C03582=1013.763,-65.159,-112.589,-25.183,25.961,-41.211
C03583=1013.760,-65.399,-112.570,-25.198,26.028,-41.179
C03584=1013.758,-65.638,-112.552,-25.214,26.096,-41.145
C03585=1013.756,-65.879,-112.533,-25.229,26.164,-41.112
C03586=1013.753,-66.119,-112.513,-25.244,26.231,-41.080
C03587=1013.750,-66.358,-112.495,-25.260,26.301,-41.045
C03588=1013.748,-66.599,-112.475,-25.275,26.369,-41.012
C03589=1013.746,-66.839,-112.456,-25.291,26.439,-40.980
C03590=1013.743,-67.080,-112.437,-25.307,26.508,-40.945
C03591=1013.740,-67.320,-112.417,-25.322,26.578,-40.911
C03592=1013.738,-67.561,-112.398,-25.338,26.649,-40.878
C03593=1013.735,-67.801,-112.379,-25.354,26.720,-40.844
C03594=1013.733,-68.042,-112.360,-25.369,26.790,-40.811
C03595=1013.730,-68.283,-112.341,-25.385,26.862,-40.776
C03596=1013.728,-68.523,-112.322,-25.401,26.933,-40.743
C03597=1013.725,-68.763,-112.303,-25.417,27.006,-40.709
C03598=1013.723,-69.004,-112.283,-25.433,27.078,-40.674
C03599=1013.720,-69.245,-112.264,-25.448,27.151,-40.640
C03600=1013.716,-69.587,-112.236,-25.471,27.255,-40.591
C03601=1013.712,-69.967,-112.206,-25.496,27.371,-40.536
C03602=1013.709,-70.208,-112.187,-25.512,27.446,-40.501
C03603=1013.707,-70.448,-112.167,-25.528,27.520,-40.467
C03604=1013.704,-70.689,-112.149,-25.544,27.595,-40.432
C03605=1013.702,-70.929,-112.130,-25.560,27.669,-40.398
C03606=1013.699,-71.170,-112.111,-25.576,27.746,-40.362
C03607=1013.696,-71.411,-112.091,-25.592,27.821,-40.328
C03608=1013.694,-71.652,-112.072,-25.608,27.897,-40.293
C03609=1013.691,-71.892,-112.053,-25.625,27.974,-40.258
C03610=1013.688,-72.132,-112.034,-25.641,28.052,-40.222
C03611=1013.686,-72.374,-112.014,-25.657,28.128,-40.186
C03612=1013.683,-72.613,-111.996,-25.673,28.205,-40.152
C03613=1013.680,-72.853,-111.976,-25.689,28.283,-40.116
C03614=1013.677,-73.094,-111.957,-25.706,28.362,-40.080
C03615=1013.675,-73.334,-111.938,-25.722,28.440,-40.044
C03616=1013.672,-73.575,-111.919,-25.738,28.519,-40.009
C03617=1013.669,-73.815,-111.900,-25.754,28.598,-39.974
C03618=1013.666,-74.054,-111.881,-25.771,28.678,-39.938
C03619=1013.663,-74.295,-111.861,-25.787,28.757,-39.902
C03620=1013.661,-74.534,-111.842,-25.803,28.838,-39.866
C03621=1013.657,-74.775,-111.823,-25.820,28.919,-39.830
C03622=1013.656,-75.014,-111.804,-25.836,28.999,-39.795
C03623=1013.652,-75.255,-111.784,-25.852,29.081,-39.759
C03624=1013.650,-75.494,-111.765,-25.869,29.162,-39.722
C03625=1013.647,-75.735,-111.746,-25.885,29.244,-39.685
C03626=1013.644,-75.974,-111.727,-25.901,29.326,-39.650
C03627=1013.640,-76.214,-111.708,-25.918,29.409,-39.614
C03628=1013.638,-76.454,-111.690,-25.934,29.492,-39.577
C03629=1013.635,-76.693,-111.670,-25.951,29.575,-39.542
C03630=1013.632,-76.932,-111.651,-25.967,29.659,-39.504
C03631=1013.630,-77.172,-111.632,-25.983,29.742,-39.468
C03632=1013.627,-77.411,-111.612,-26.000,29.827,-39.432
C03633=1013.623,-77.650,-111.594,-26.016,29.911,-39.395
C03634=1013.620,-77.889,-111.574,-26.033,29.996,-39.358
C03635=1013.618,-78.129,-111.556,-26.049,30.081,-39.322
C03636=1013.614,-78.367,-111.536,-26.066,30.167,-39.286
C03637=1013.611,-78.606,-111.517,-26.082,30.252,-39.249
C03638=1013.608,-78.844,-111.498,-26.099,30.339,-39.212
C03639=1013.605,-79.083,-111.479,-26.115,30.425,-39.176
C03640=1013.602,-79.321,-111.460,-26.132,30.511,-39.139
C03641=1013.599,-79.559,-111.441,-26.148,30.598,-39.102
C03642=1013.597,-79.798,-111.422,-26.165,30.686,-39.066
C03643=1013.594,-80.036,-111.403,-26.181,30.772,-39.029
C03644=1013.591,-80.274,-111.384,-26.197,30.861,-38.991
C03645=1013.587,-80.511,-111.365,-26.214,30.949,-38.955
C03646=1013.585,-80.748,-111.346,-26.230,31.038,-38.918
C03647=1013.582,-80.985,-111.327,-26.247,31.125,-38.881
C03648=1013.578,-81.220,-111.308,-26.263,31.215,-38.844
C03649=1013.576,-81.457,-111.289,-26.279,31.303,-38.808
C03650=1013.573,-81.694,-111.270,-26.296,31.393,-38.772
C03651=1013.570,-81.930,-111.251,-26.312,31.483,-38.734
C03652=1013.567,-82.168,-111.233,-26.329,31.573,-38.698
C03653=1013.564,-82.405,-111.213,-26.345,31.664,-38.660
C03654=1013.560,-82.642,-111.195,-26.361,31.755,-38.624
C03655=1013.558,-82.878,-111.176,-26.378,31.846,-38.587
C03656=1013.554,-83.113,-111.157,-26.394,31.937,-38.549
C03657=1013.552,-83.350,-111.138,-26.411,32.029,-38.513
C03658=1013.548,-83.586,-111.119,-26.427,32.121,-38.476
C03659=1013.545,-83.821,-111.101,-26.443,32.213,-38.439
C03660=1013.542,-84.054,-111.082,-26.460,32.304,-38.402
C03661=1013.539,-84.286,-111.063,-26.476,32.396,-38.366
C03662=1013.536,-84.519,-111.044,-26.492,32.488,-38.329
C03663=1013.533,-84.759,-111.025,-26.509,32.584,-38.291
C03664=1013.529,-85.016,-111.004,-26.526,32.686,-38.252
C03665=1013.526,-85.291,-110.983,-26.545,32.796,-38.208
C03666=1013.523,-85.531,-110.963,-26.562,32.893,-38.169
C03667=1013.518,-85.858,-110.937,-26.585,33.025,-38.119
C03668=1013.514,-86.127,-110.915,-26.603,33.135,-38.077
C03669=1013.510,-86.378,-110.895,-26.621,33.237,-38.038
C03670=1013.508,-86.612,-110.877,-26.637,33.332,-38.000
C03671=1013.505,-86.843,-110.858,-26.653,33.428,-37.963
C03672=1013.502,-87.073,-110.840,-26.669,33.523,-37.927
C03673=1013.499,-87.296,-110.822,-26.685,33.614,-37.892
C03674=1013.495,-87.515,-110.804,-26.700,33.705,-37.858
C03675=1013.493,-87.735,-110.787,-26.715,33.797,-37.822
C03676=1013.489,-87.950,-110.769,-26.730,33.886,-37.788
C03677=1013.486,-88.167,-110.753,-26.745,33.978,-37.754
C03678=1013.484,-88.393,-110.735,-26.761,34.073,-37.719
C03679=1013.480,-88.619,-110.716,-26.776,34.168,-37.683
C03680=1013.477,-88.853,-110.697,-26.792,34.267,-37.646
C03681=1013.474,-89.120,-110.676,-26.811,34.380,-37.604
C03682=1013.470,-89.416,-110.652,-26.831,34.506,-37.557
C03683=1013.466,-89.724,-110.627,-26.853,34.638,-37.507
C03684=1013.461,-90.025,-110.603,-26.873,34.768,-37.461
C03685=1013.455,-90.431,-110.571,-26.901,34.943,-37.396
C03686=1013.451,-90.700,-110.549,-26.920,35.060,-37.354
C03687=1013.447,-90.997,-110.525,-26.940,35.190,-37.306
C03688=1013.443,-91.247,-110.505,-26.957,35.298,-37.269
C03689=1013.440,-91.478,-110.486,-26.973,35.401,-37.231
C03690=1013.437,-91.710,-110.467,-26.989,35.502,-37.195
C03691=1013.434,-91.941,-110.449,-27.005,35.604,-37.159
C03692=1013.431,-92.172,-110.430,-27.021,35.707,-37.122
C03693=1013.428,-92.403,-110.412,-27.036,35.809,-37.086
C03694=1013.424,-92.633,-110.393,-27.052,35.911,-37.049
C03695=1013.421,-92.864,-110.375,-27.068,36.014,-37.014
C03696=1013.418,-93.095,-110.356,-27.084,36.118,-36.978
C03697=1013.414,-93.324,-110.338,-27.099,36.220,-36.941
C03698=1013.411,-93.553,-110.319,-27.115,36.324,-36.905
C03699=1013.408,-93.783,-110.300,-27.130,36.427,-36.870
C03700=1013.405,-94.011,-110.282,-27.146,36.531,-36.835
C03701=1013.401,-94.240,-110.263,-27.161,36.635,-36.799
C03702=1013.398,-94.468,-110.245,-27.177,36.738,-36.763
C03703=1013.395,-94.695,-110.227,-27.192,36.843,-36.728
C03704=1013.391,-94.922,-110.208,-27.208,36.947,-36.692
C03705=1013.387,-95.149,-110.190,-27.223,37.051,-36.657
C03706=1013.385,-95.375,-110.172,-27.238,37.156,-36.622
C03707=1013.381,-95.601,-110.153,-27.253,37.259,-36.587
C03708=1013.378,-95.826,-110.135,-27.269,37.365,-36.551
C03709=1013.375,-96.052,-110.117,-27.284,37.469,-36.516
C03710=1013.372,-96.276,-110.100,-27.299,37.574,-36.481
C03711=1013.368,-96.501,-110.081,-27.314,37.678,-36.447
C03712=1013.365,-96.725,-110.062,-27.329,37.784,-36.413
C03713=1013.362,-96.949,-110.045,-27.344,37.888,-36.379
C03714=1013.358,-97.173,-110.026,-27.359,37.995,-36.344
C03715=1013.355,-97.397,-110.008,-27.374,38.100,-36.310
C03716=1013.352,-97.620,-109.990,-27.389,38.207,-36.275
C03717=1013.349,-97.844,-109.973,-27.403,38.312,-36.242
C03718=1013.345,-98.067,-109.955,-27.418,38.419,-36.207
C03719=1013.340,-98.468,-109.922,-27.445,38.610,-36.146
C03720=1013.335,-98.738,-109.900,-27.463,38.739,-36.104
C03721=1013.332,-98.962,-109.882,-27.478,38.848,-36.070
C03722=1013.329,-99.186,-109.864,-27.492,38.955,-36.036
C03723=1013.326,-99.410,-109.846,-27.507,39.064,-36.001
C03724=1013.322,-99.635,-109.827,-27.522,39.173,-35.967
C03725=1013.319,-99.859,-109.809,-27.537,39.283,-35.933
C03726=1013.316,-100.085,-109.791,-27.552,39.393,-35.900
C03727=1013.312,-100.310,-109.773,-27.567,39.504,-35.865
C03728=1013.309,-100.536,-109.754,-27.581,39.613,-35.831
C03729=1013.305,-100.762,-109.736,-27.596,39.725,-35.797
C03730=1013.302,-100.989,-109.717,-27.611,39.836,-35.763
C03731=1013.299,-101.216,-109.700,-27.626,39.949,-35.728
C03732=1013.295,-101.443,-109.681,-27.641,40.061,-35.695
C03733=1013.292,-101.671,-109.662,-27.656,40.174,-35.660
C03734=1013.288,-101.899,-109.643,-27.670,40.288,-35.627
C03735=1013.285,-102.128,-109.624,-27.685,40.402,-35.592
C03736=1013.282,-102.356,-109.607,-27.700,40.517,-35.557
C03737=1013.278,-102.585,-109.588,-27.715,40.632,-35.524
C03738=1013.275,-102.814,-109.569,-27.730,40.746,-35.490
C03739=1013.271,-103.044,-109.551,-27.745,40.862,-35.456
C03740=1013.268,-103.274,-109.532,-27.760,40.979,-35.422
C03741=1013.265,-103.503,-109.513,-27.774,41.095,-35.388
C03742=1013.261,-103.733,-109.494,-27.789,41.212,-35.354
C03743=1013.257,-103.964,-109.475,-27.804,41.329,-35.321
C03744=1013.253,-104.194,-109.457,-27.819,41.447,-35.287
C03745=1013.251,-104.425,-109.438,-27.834,41.565,-35.253
C03746=1013.247,-104.655,-109.420,-27.848,41.683,-35.219
C03747=1013.243,-104.887,-109.400,-27.863,41.802,-35.187
C03748=1013.241,-105.118,-109.381,-27.878,41.921,-35.152
C03749=1013.236,-105.349,-109.362,-27.893,42.041,-35.119
C03750=1013.233,-105.580,-109.344,-27.907,42.161,-35.086
C03751=1013.230,-105.812,-109.324,-27.922,42.281,-35.052
C03752=1013.226,-106.043,-109.306,-27.937,42.402,-35.019
C03753=1013.222,-106.275,-109.287,-27.952,42.522,-34.986
C03754=1013.219,-106.510,-109.268,-27.966,42.645,-34.953
C03755=1013.216,-106.752,-109.248,-27.982,42.772,-34.918
C03756=1013.212,-107.005,-109.227,-27.998,42.904,-34.883
C03757=1013.207,-107.267,-109.206,-28.014,43.043,-34.846
C03758=1013.204,-107.537,-109.184,-28.031,43.186,-34.806
C03759=1013.199,-107.812,-109.161,-28.049,43.332,-34.767
C03760=1013.195,-108.089,-109.138,-28.066,43.478,-34.728
C03761=1013.191,-108.362,-109.117,-28.083,43.625,-34.690
C03762=1013.187,-108.631,-109.095,-28.100,43.769,-34.652
C03763=1013.183,-108.891,-109.074,-28.116,43.908,-34.616
C03764=1013.180,-109.142,-109.053,-28.132,44.042,-34.581
C03765=1013.176,-109.383,-109.033,-28.147,44.172,-34.548
C03766=1013.170,-109.734,-109.003,-28.169,44.360,-34.500
C03767=1013.165,-110.079,-108.975,-28.190,44.548,-34.453
C03768=1013.162,-110.311,-108.957,-28.205,44.674,-34.422
C03769=1013.158,-110.542,-108.938,-28.219,44.800,-34.391
C03770=1013.155,-110.773,-108.919,-28.233,44.927,-34.359
C03771=1013.151,-111.005,-108.900,-28.248,45.053,-34.328
C03772=1013.148,-111.236,-108.881,-28.262,45.180,-34.296
C03773=1013.144,-111.468,-108.862,-28.276,45.307,-34.265
C03774=1013.140,-111.698,-108.843,-28.290,45.433,-34.235
C03775=1013.137,-111.930,-108.823,-28.305,45.561,-34.204
C03776=1013.134,-112.162,-108.805,-28.319,45.690,-34.174
C03777=1013.129,-112.393,-108.786,-28.333,45.818,-34.142
C03778=1013.126,-112.624,-108.767,-28.347,45.947,-34.112
C03779=1013.123,-112.855,-108.747,-28.362,46.074,-34.082
C03780=1013.119,-113.087,-108.729,-28.376,46.205,-34.052
C03781=1013.116,-113.318,-108.709,-28.390,46.334,-34.021
C03782=1013.112,-113.549,-108.691,-28.404,46.462,-33.992
C03783=1013.109,-113.781,-108.671,-28.418,46.593,-33.962
C03784=1013.106,-114.011,-108.652,-28.433,46.723,-33.932
C03785=1013.102,-114.243,-108.633,-28.447,46.853,-33.903
C03786=1013.098,-114.474,-108.614,-28.461,46.984,-33.872
C03787=1013.095,-114.705,-108.595,-28.475,47.115,-33.843
C03788=1013.092,-114.937,-108.576,-28.489,47.247,-33.814
C03789=1013.088,-115.168,-108.557,-28.503,47.378,-33.785
C03790=1013.085,-115.399,-108.538,-28.517,47.510,-33.756
C03791=1013.081,-115.630,-108.519,-28.531,47.641,-33.728
C03792=1013.077,-115.861,-108.499,-28.545,47.773,-33.699
C03793=1013.074,-116.093,-108.481,-28.559,47.905,-33.670
C03794=1013.071,-116.324,-108.461,-28.573,48.038,-33.642
C03795=1013.066,-116.555,-108.442,-28.587,48.171,-33.614
C03796=1013.064,-116.786,-108.424,-28.601,48.304,-33.584
C03797=1013.060,-117.017,-108.404,-28.615,48.437,-33.557
C03798=1013.057,-117.248,-108.385,-28.629,48.570,-33.530
C03799=1013.053,-117.479,-108.365,-28.643,48.704,-33.501
C03800=1013.050,-117.711,-108.346,-28.657,48.837,-33.474
C03801=1013.046,-117.942,-108.328,-28.671,48.972,-33.446
C03802=1013.043,-118.173,-108.308,-28.685,49.107,-33.419
C03803=1013.040,-118.404,-108.290,-28.699,49.240,-33.393
C03804=1013.036,-118.635,-108.270,-28.713,49.376,-33.366
C03805=1013.033,-118.867,-108.251,-28.727,49.510,-33.339
C03806=1013.029,-119.097,-108.232,-28.741,49.646,-33.311
C03807=1013.023,-119.517,-108.197,-28.767,49.892,-33.263
C03808=1013.019,-119.791,-108.174,-28.783,50.052,-33.234
C03809=1013.016,-120.021,-108.155,-28.797,50.188,-33.207
C03810=1013.012,-120.253,-108.135,-28.811,50.324,-33.182
C03811=1013.009,-120.484,-108.117,-28.825,50.460,-33.156
C03812=1013.005,-120.715,-108.098,-28.839,50.597,-33.130
C03813=1013.001,-120.946,-108.078,-28.853,50.734,-33.104
C03814=1012.998,-121.177,-108.059,-28.867,50.871,-33.080
C03815=1012.995,-121.408,-108.039,-28.881,51.009,-33.055
C03816=1012.992,-121.639,-108.021,-28.895,51.146,-33.030
C03817=1012.988,-121.871,-108.001,-28.909,51.283,-33.005
C03818=1012.985,-122.101,-107.982,-28.923,51.421,-32.981
C03819=1012.982,-122.333,-107.962,-28.937,51.560,-32.957
C03820=1012.978,-122.563,-107.944,-28.951,51.697,-32.933
C03821=1012.974,-122.794,-107.924,-28.965,51.836,-32.909
C03822=1012.971,-123.025,-107.906,-28.979,51.974,-32.885
C03823=1012.968,-123.257,-107.886,-28.993,52.113,-32.862
C03824=1012.965,-123.487,-107.867,-29.007,52.253,-32.839
C03825=1012.962,-123.718,-107.848,-29.021,52.392,-32.815
C03826=1012.958,-123.949,-107.828,-29.035,52.531,-32.792
C03827=1012.955,-124.180,-107.809,-29.050,52.671,-32.770
C03828=1012.951,-124.411,-107.789,-29.064,52.811,-32.747
C03829=1012.949,-124.642,-107.771,-29.078,52.950,-32.725
C03830=1012.945,-124.874,-107.751,-29.092,53.091,-32.702
C03831=1012.942,-125.104,-107.732,-29.107,53.231,-32.681
C03832=1012.938,-125.336,-107.712,-29.121,53.372,-32.658
C03833=1012.935,-125.566,-107.693,-29.135,53.512,-32.638
C03834=1012.932,-125.797,-107.674,-29.149,53.654,-32.616
C03835=1012.929,-126.028,-107.654,-29.164,53.795,-32.595
C03836=1012.926,-126.259,-107.635,-29.178,53.936,-32.573
C03837=1012.922,-126.490,-107.615,-29.193,54.078,-32.552
C03838=1012.919,-126.721,-107.596,-29.207,54.219,-32.532
C03839=1012.916,-126.952,-107.578,-29.221,54.362,-32.511
C03840=1012.913,-127.183,-107.558,-29.236,54.504,-32.491
C03841=1012.910,-127.414,-107.539,-29.251,54.646,-32.472
C03842=1012.906,-127.645,-107.519,-29.265,54.789,-32.451
C03843=1012.903,-127.876,-107.500,-29.280,54.931,-32.432
C03844=1012.900,-128.106,-107.481,-29.294,55.074,-32.412
C03845=1012.896,-128.337,-107.461,-29.309,55.218,-32.393
C03846=1012.890,-128.749,-107.427,-29.336,55.474,-32.360
C03847=1012.886,-129.030,-107.403,-29.354,55.649,-32.337
C03848=1012.883,-129.261,-107.384,-29.369,55.792,-32.319
C03849=1012.880,-129.491,-107.365,-29.384,55.936,-32.301
C03850=1012.877,-129.722,-107.345,-29.399,56.081,-32.283
C03851=1012.874,-129.953,-107.326,-29.414,56.225,-32.266
C03852=1012.871,-130.184,-107.307,-29.429,56.370,-32.248
C03853=1012.867,-130.415,-107.287,-29.444,56.515,-32.230
C03854=1012.865,-130.646,-107.267,-29.460,56.659,-32.215
C03855=1012.862,-130.876,-107.248,-29.475,56.805,-32.198
C03856=1012.858,-131.108,-107.228,-29.490,56.950,-32.182
C03857=1012.855,-131.339,-107.210,-29.506,57.095,-32.165
C03858=1012.852,-131.570,-107.191,-29.521,57.242,-32.148
C03859=1012.849,-131.800,-107.171,-29.537,57.388,-32.133
C03860=1012.846,-132.031,-107.152,-29.553,57.534,-32.118
C03861=1012.843,-132.262,-107.132,-29.568,57.680,-32.102
C03862=1012.840,-132.493,-107.113,-29.585,57.827,-32.089
C03863=1012.837,-132.724,-107.093,-29.600,57.974,-32.073
C03864=1012.834,-132.955,-107.074,-29.616,58.121,-32.059
C03865=1012.830,-133.185,-107.055,-29.633,58.268,-32.045
C03866=1012.828,-133.416,-107.035,-29.649,58.415,-32.031
C03867=1012.825,-133.647,-107.016,-29.665,58.563,-32.017
C03868=1012.821,-133.878,-106.996,-29.682,58.710,-32.004
C03869=1012.818,-134.109,-106.977,-29.698,58.858,-31.992
C03870=1013.073,-134.133,-107.391,-28.594,48.007,-33.824
C03871=1013.076,-133.902,-107.411,-28.577,47.850,-33.859
C03872=1013.080,-133.672,-107.430,-28.560,47.694,-33.892
C03873=1013.084,-133.441,-107.449,-28.544,47.538,-33.928
C03874=1013.089,-133.210,-107.468,-28.527,47.382,-33.964
C03875=1013.093,-132.979,-107.487,-28.510,47.227,-33.999
C03876=1013.096,-132.748,-107.506,-28.493,47.070,-34.035
C03877=1013.101,-132.517,-107.525,-28.476,46.914,-34.071
C03878=1013.105,-132.286,-107.544,-28.458,46.759,-34.107
C03879=1013.109,-132.055,-107.563,-28.441,46.604,-34.143
C03880=1013.114,-131.824,-107.582,-28.424,46.448,-34.181
C03881=1013.118,-131.594,-107.600,-28.407,46.294,-34.218
C03882=1013.121,-131.363,-107.620,-28.390,46.139,-34.254
C03883=1013.126,-131.132,-107.639,-28.373,45.985,-34.291
C03884=1013.130,-130.901,-107.658,-28.355,45.831,-34.329
C03885=1013.134,-130.670,-107.677,-28.338,45.677,-34.367
C03886=1013.138,-130.439,-107.696,-28.321,45.524,-34.405
C03887=1013.143,-130.208,-107.715,-28.303,45.371,-34.442
C03888=1013.147,-129.977,-107.734,-28.286,45.217,-34.481
C03889=1013.151,-129.746,-107.753,-28.268,45.064,-34.520
C03890=1013.155,-129.516,-107.771,-28.251,44.911,-34.558
C03891=1013.159,-129.285,-107.791,-28.233,44.759,-34.598
C03892=1013.163,-129.054,-107.810,-28.215,44.606,-34.636
C03893=1013.171,-128.685,-107.841,-28.187,44.364,-34.699
C03894=1013.176,-128.361,-107.867,-28.162,44.152,-34.754
C03895=1013.180,-128.130,-107.886,-28.144,43.999,-34.795
C03896=1013.184,-127.899,-107.905,-28.127,43.849,-34.834
C03897=1013.189,-127.668,-107.924,-28.109,43.698,-34.875
C03898=1013.193,-127.437,-107.943,-28.091,43.548,-34.916
C03899=1013.198,-127.207,-107.962,-28.073,43.398,-34.957
C03900=1013.202,-126.976,-107.981,-28.055,43.247,-34.998
C03901=1013.206,-126.745,-108.000,-28.037,43.098,-35.039
C03902=1013.210,-126.514,-108.018,-28.018,42.948,-35.081
C03903=1013.214,-126.283,-108.037,-28.000,42.798,-35.122
C03904=1013.219,-126.052,-108.056,-27.982,42.649,-35.163
C03905=1013.223,-125.821,-108.074,-27.964,42.500,-35.206
C03906=1013.227,-125.590,-108.093,-27.945,42.352,-35.248
C03907=1013.232,-125.359,-108.112,-27.927,42.203,-35.289
C03908=1013.236,-125.128,-108.132,-27.908,42.056,-35.332
C03909=1013.240,-124.897,-108.150,-27.890,41.907,-35.375
C03910=1013.244,-124.666,-108.169,-27.871,41.759,-35.417
C03911=1013.249,-124.435,-108.188,-27.852,41.612,-35.461
C03912=1013.253,-124.204,-108.207,-27.833,41.464,-35.504
C03913=1013.258,-123.973,-108.225,-27.815,41.318,-35.547
C03914=1013.262,-123.742,-108.244,-27.796,41.171,-35.591
C03915=1013.267,-123.511,-108.263,-27.777,41.025,-35.634
C03916=1013.271,-123.280,-108.282,-27.758,40.879,-35.679
C03917=1013.275,-123.049,-108.301,-27.739,40.733,-35.722
C03918=1013.279,-122.818,-108.319,-27.720,40.587,-35.766
C03919=1013.283,-122.587,-108.338,-27.701,40.441,-35.812
C03920=1013.288,-122.356,-108.357,-27.681,40.296,-35.856
C03921=1013.292,-122.125,-108.376,-27.662,40.151,-35.900
C03922=1013.296,-121.894,-108.395,-27.643,40.006,-35.946
C03923=1013.300,-121.663,-108.413,-27.623,39.862,-35.991
C03924=1013.305,-121.432,-108.431,-27.604,39.718,-36.037
C03925=1013.310,-121.201,-108.450,-27.584,39.573,-36.082
C03926=1013.314,-120.970,-108.469,-27.565,39.430,-36.127
C03927=1013.318,-120.738,-108.488,-27.545,39.287,-36.173
C03928=1013.323,-120.507,-108.507,-27.525,39.144,-36.219
C03929=1013.327,-120.276,-108.526,-27.505,39.000,-36.265
C03930=1013.331,-120.045,-108.545,-27.486,38.858,-36.311
C03931=1013.335,-119.814,-108.563,-27.466,38.715,-36.359
C03932=1013.340,-119.569,-108.582,-27.444,38.565,-36.407
C03933=1013.344,-119.353,-108.600,-27.425,38.432,-36.452
C03934=1013.348,-119.121,-108.618,-27.405,38.290,-36.498
C03935=1013.353,-118.890,-108.637,-27.385,38.149,-36.546
C03936=1013.357,-118.659,-108.656,-27.365,38.008,-36.593
C03937=1013.361,-118.428,-108.675,-27.344,37.867,-36.641
C03938=1013.366,-118.197,-108.694,-27.324,37.726,-36.689
C03939=1013.371,-117.966,-108.712,-27.304,37.586,-36.736
C03940=1013.375,-117.734,-108.730,-27.283,37.446,-36.784
C03941=1013.379,-117.503,-108.749,-27.262,37.306,-36.833
C03942=1013.384,-117.272,-108.768,-27.242,37.166,-36.881
C03943=1013.388,-117.041,-108.787,-27.221,37.027,-36.930
C03944=1013.392,-116.810,-108.806,-27.200,36.887,-36.978
C03945=1013.396,-116.578,-108.824,-27.179,36.749,-37.026
C03946=1013.401,-116.347,-108.842,-27.158,36.611,-37.075
C03947=1013.406,-116.116,-108.861,-27.137,36.473,-37.124
C03948=1013.410,-115.885,-108.880,-27.116,36.335,-37.173
C03949=1013.414,-115.654,-108.899,-27.095,36.197,-37.223
C03950=1013.418,-115.422,-108.917,-27.073,36.059,-37.272
C03951=1013.423,-115.191,-108.936,-27.052,35.922,-37.322
C03952=1013.427,-114.960,-108.954,-27.031,35.785,-37.372
C03953=1013.432,-114.729,-108.973,-27.009,35.649,-37.422
C03954=1013.436,-114.497,-108.991,-26.988,35.512,-37.472
C03955=1013.440,-114.266,-109.010,-26.966,35.376,-37.523
C03956=1013.444,-114.035,-109.028,-26.944,35.241,-37.573
C03957=1013.449,-113.804,-109.047,-26.923,35.105,-37.623
C03958=1013.453,-113.572,-109.065,-26.901,34.970,-37.674
C03959=1013.458,-113.341,-109.084,-26.879,34.835,-37.726
C03960=1013.462,-113.110,-109.102,-26.857,34.700,-37.777
C03961=1013.466,-112.878,-109.121,-26.835,34.566,-37.828
C03962=1013.470,-112.647,-109.140,-26.813,34.432,-37.879
C03963=1013.474,-112.416,-109.158,-26.791,34.299,-37.930
C03964=1013.480,-112.185,-109.176,-26.768,34.165,-37.981
C03965=1013.484,-111.953,-109.195,-26.746,34.031,-38.034
C03966=1013.488,-111.722,-109.213,-26.723,33.899,-38.085
C03967=1013.492,-111.491,-109.232,-26.701,33.766,-38.138
C03968=1013.496,-111.259,-109.250,-26.678,33.635,-38.189
C03969=1013.501,-111.028,-109.269,-26.656,33.502,-38.241
C03970=1013.505,-110.797,-109.287,-26.633,33.372,-38.293
C03971=1013.509,-110.565,-109.305,-26.611,33.240,-38.346
C03972=1013.513,-110.351,-109.322,-26.589,33.119,-38.395
C03973=1013.517,-110.137,-109.340,-26.568,32.999,-38.443
C03974=1013.522,-109.871,-109.361,-26.542,32.849,-38.503
C03975=1013.526,-109.639,-109.379,-26.519,32.719,-38.556
C03976=1013.531,-109.406,-109.397,-26.496,32.588,-38.610
C03977=1013.535,-109.165,-109.416,-26.472,32.454,-38.664
C03978=1013.540,-108.915,-109.437,-26.447,32.315,-38.720
C03979=1013.545,-108.654,-109.458,-26.421,32.171,-38.781
C03980=1013.550,-108.386,-109.478,-26.394,32.022,-38.843
C03981=1013.555,-108.112,-109.500,-26.366,31.871,-38.907
C03982=1013.560,-107.835,-109.522,-26.338,31.720,-38.971
C03983=1013.565,-107.560,-109.545,-26.310,31.568,-39.036
C03984=1013.570,-107.290,-109.566,-26.282,31.421,-39.099
C03985=1013.575,-107.028,-109.587,-26.256,31.278,-39.161
C03986=1013.580,-106.775,-109.606,-26.230,31.141,-39.219
C03987=1013.584,-106.533,-109.626,-26.205,31.010,-39.275
C03988=1013.588,-106.298,-109.644,-26.181,30.883,-39.330
C03989=1013.593,-106.067,-109.663,-26.157,30.758,-39.385
C03990=1013.597,-105.835,-109.682,-26.133,30.634,-39.438
C03991=1013.601,-105.604,-109.699,-26.109,30.510,-39.493
C03992=1013.605,-105.372,-109.718,-26.085,30.387,-39.547
C03993=1013.610,-105.140,-109.736,-26.061,30.263,-39.602
C03994=1013.614,-104.909,-109.755,-26.036,30.141,-39.657
C03995=1013.618,-104.679,-109.772,-26.012,30.020,-39.711
C03996=1013.623,-104.448,-109.791,-25.988,29.898,-39.766
C03997=1013.626,-104.217,-109.809,-25.964,29.777,-39.821
C03998=1013.630,-103.987,-109.827,-25.940,29.655,-39.875
C03999=1013.634,-103.757,-109.846,-25.915,29.535,-39.930
C04000=1013.639,-103.527,-109.864,-25.891,29.415,-39.985
C04001=1013.643,-103.297,-109.882,-25.867,29.296,-40.040
C04002=1013.647,-103.066,-109.900,-25.842,29.177,-40.095
C04003=1013.651,-102.837,-109.918,-25.817,29.057,-40.150
C04004=1013.656,-102.607,-109.936,-25.793,28.940,-40.205
C04005=1013.660,-102.379,-109.955,-25.769,28.822,-40.260
C04006=1013.664,-102.149,-109.972,-25.744,28.705,-40.315
C04007=1013.667,-101.921,-109.990,-25.719,28.588,-40.370
C04008=1013.672,-101.693,-110.008,-25.695,28.472,-40.424
C04009=1013.676,-101.465,-110.026,-25.670,28.356,-40.480
C04010=1013.681,-101.238,-110.044,-25.646,28.241,-40.535
C04011=1013.684,-101.011,-110.062,-25.621,28.126,-40.590
C04012=1013.688,-100.785,-110.080,-25.596,28.013,-40.644
C04013=1013.692,-100.559,-110.097,-25.572,27.899,-40.700
C04014=1013.696,-100.332,-110.115,-25.547,27.786,-40.754
C04015=1013.700,-100.107,-110.133,-25.523,27.673,-40.809
C04016=1013.704,-99.881,-110.151,-25.498,27.562,-40.863
C04017=1013.708,-99.657,-110.168,-25.473,27.450,-40.918
C04018=1013.713,-99.373,-110.190,-25.442,27.310,-40.986
C04019=1013.720,-98.984,-110.221,-25.399,27.119,-41.081
C04020=1013.724,-98.760,-110.238,-25.375,27.008,-41.136
C04021=1013.728,-98.537,-110.256,-25.350,26.900,-41.190
C04022=1013.731,-98.312,-110.274,-25.325,26.790,-41.245
C04023=1013.735,-98.089,-110.292,-25.300,26.682,-41.299
C04024=1013.739,-97.865,-110.309,-25.276,26.574,-41.354
C04025=1013.744,-97.642,-110.327,-25.251,26.466,-41.408
C04026=1013.747,-97.419,-110.344,-25.226,26.358,-41.463
C04027=1013.751,-97.195,-110.361,-25.201,26.251,-41.518
C04028=1013.754,-96.971,-110.379,-25.176,26.144,-41.574
C04029=1013.759,-96.747,-110.397,-25.151,26.037,-41.627
C04030=1013.763,-96.523,-110.414,-25.125,25.931,-41.683
C04031=1013.767,-96.298,-110.432,-25.100,25.825,-41.738
C04032=1013.770,-96.073,-110.449,-25.075,25.719,-41.793
C04033=1013.774,-95.849,-110.467,-25.050,25.613,-41.848
C04034=1013.778,-95.622,-110.484,-25.024,25.507,-41.904
C04035=1013.782,-95.397,-110.502,-24.999,25.402,-41.959
C04036=1013.786,-95.171,-110.520,-24.973,25.296,-42.016
C04037=1013.790,-94.944,-110.537,-24.947,25.191,-42.071
C04038=1013.793,-94.716,-110.555,-24.921,25.086,-42.128
C04039=1013.797,-94.489,-110.572,-24.896,24.980,-42.183
C04040=1013.801,-94.261,-110.591,-24.870,24.875,-42.241
C04041=1013.805,-94.033,-110.609,-24.844,24.771,-42.296
C04042=1013.809,-93.804,-110.627,-24.818,24.667,-42.352
C04043=1013.813,-93.574,-110.644,-24.791,24.562,-42.410
C04044=1013.817,-93.345,-110.662,-24.765,24.458,-42.466
C04045=1013.820,-93.116,-110.680,-24.739,24.355,-42.523
C04046=1013.824,-92.886,-110.698,-24.713,24.251,-42.579
C04047=1013.828,-92.655,-110.716,-24.686,24.147,-42.636
C04048=1013.832,-92.424,-110.735,-24.659,24.044,-42.695
C04049=1013.836,-92.194,-110.752,-24.633,23.941,-42.752
C04050=1013.839,-91.963,-110.770,-24.607,23.839,-42.808
C04051=1013.843,-91.731,-110.788,-24.580,23.736,-42.865
C04052=1013.847,-91.500,-110.806,-24.553,23.634,-42.923
C04053=1013.851,-91.269,-110.825,-24.526,23.532,-42.981
C04054=1013.855,-91.018,-110.844,-24.498,23.423,-43.041
C04055=1013.859,-90.722,-110.867,-24.463,23.293,-43.117
C04056=1013.864,-90.453,-110.889,-24.432,23.175,-43.183
C04057=1013.870,-90.047,-110.919,-24.385,23.001,-43.283
C04058=1013.876,-89.746,-110.943,-24.350,22.872,-43.358
C04059=1013.880,-89.438,-110.967,-24.314,22.739,-43.434
C04060=1013.885,-89.142,-110.990,-24.279,22.614,-43.508
C04061=1013.889,-88.874,-111.011,-24.248,22.500,-43.574
C04062=1013.893,-88.641,-111.029,-24.221,22.402,-43.632
C04063=1013.897,-88.414,-111.047,-24.194,22.306,-43.688
C04064=1013.900,-88.188,-111.065,-24.168,22.211,-43.744
C04065=1013.904,-87.971,-111.082,-24.142,22.121,-43.798
C04066=1013.921,-86.931,-111.162,-24.009,21.652,-44.080
C04067=1013.925,-86.605,-111.188,-24.010,21.651,-44.075
C04068=1013.931,-86.261,-111.214,-24.011,21.651,-44.069
C04069=1013.934,-86.030,-111.232,-24.011,21.650,-44.065
C04070=1013.938,-85.785,-111.251,-24.012,21.650,-44.062
C04071=1013.941,-85.529,-111.271,-24.012,21.649,-44.060
C04072=1013.945,-85.276,-111.291,-24.012,21.650,-44.056
C04073=1013.949,-85.034,-111.309,-24.013,21.649,-44.053
C04074=1013.952,-84.812,-111.327,-24.013,21.649,-44.049
C04075=1013.958,-84.404,-111.359,-24.014,21.648,-44.043
C04076=1013.964,-84.005,-111.390,-24.015,21.648,-44.036
C04077=1013.970,-83.604,-111.421,-24.016,21.647,-44.031
C04078=1013.977,-83.204,-111.452,-24.016,21.646,-44.025
C04079=1013.982,-82.801,-111.484,-24.017,21.645,-44.019
C04080=1013.988,-82.399,-111.515,-24.018,21.644,-44.014
C04081=1013.993,-81.997,-111.546,-24.019,21.644,-44.007
C04082=1013.999,-81.593,-111.578,-24.020,21.643,-44.001
C04083=1014.004,-81.189,-111.609,-24.020,21.643,-43.995
C04084=1014.010,-80.784,-111.641,-24.021,21.642,-43.990
C04085=1014.015,-80.379,-111.672,-24.022,21.641,-43.984
C04086=1014.021,-79.973,-111.704,-24.023,21.641,-43.977
C04087=1014.026,-79.567,-111.736,-24.023,21.640,-43.972
C04088=1014.032,-79.160,-111.767,-24.024,21.639,-43.966
C04089=1014.038,-78.753,-111.799,-24.025,21.638,-43.960
C04090=1014.043,-78.345,-111.830,-24.026,21.638,-43.953
C04091=1014.048,-77.937,-111.863,-24.027,21.637,-43.948
C04092=1014.053,-77.529,-111.894,-24.027,21.637,-43.942
C04093=1014.059,-77.120,-111.926,-24.028,21.636,-43.936
C04094=1014.063,-76.710,-111.958,-24.029,21.636,-43.929
C04095=1014.069,-76.301,-111.990,-24.030,21.635,-43.924
C04096=1014.074,-75.891,-112.022,-24.031,21.634,-43.918
C04097=1014.079,-75.481,-112.053,-24.031,21.633,-43.912
C04098=1014.085,-75.072,-112.086,-24.032,21.633,-43.905
C04099=1014.089,-74.660,-112.118,-24.033,21.632,-43.900
C04100=1014.094,-74.250,-112.150,-24.034,21.632,-43.894
C04101=1014.099,-73.839,-112.183,-24.034,21.631,-43.888
C04102=1014.104,-73.429,-112.215,-24.035,21.631,-43.881
C04103=1014.109,-73.018,-112.246,-24.036,21.630,-43.876
C04104=1014.114,-72.607,-112.278,-24.037,21.629,-43.870
C04105=1014.118,-72.196,-112.311,-24.038,21.628,-43.865
C04106=1014.123,-71.785,-112.343,-24.039,21.627,-43.857
C04107=1014.128,-71.374,-112.376,-24.039,21.626,-43.851
C04108=1014.132,-70.962,-112.407,-24.040,21.626,-43.846
C04109=1014.137,-70.552,-112.440,-24.041,21.625,-43.839
C04110=1014.141,-70.141,-112.471,-24.042,21.625,-43.833
C04111=1014.146,-69.730,-112.504,-24.042,21.624,-43.827
C04112=1014.150,-69.318,-112.536,-24.043,21.623,-43.822
C04113=1014.155,-68.908,-112.568,-24.044,21.623,-43.815
C04114=1014.159,-68.498,-112.601,-24.045,21.622,-43.809
C04115=1014.163,-68.086,-112.633,-24.046,21.621,-43.804
C04116=1014.167,-67.677,-112.665,-24.046,21.621,-43.798
C04117=1014.171,-67.266,-112.698,-24.047,21.620,-43.791
C04118=1014.176,-66.856,-112.729,-24.048,21.620,-43.785
C04119=1014.180,-66.448,-112.761,-24.049,21.619,-43.780
C04120=1014.184,-66.037,-112.794,-24.049,21.618,-43.774
C04121=1014.188,-65.629,-112.826,-24.050,21.617,-43.768
C04122=1014.192,-65.221,-112.858,-24.051,21.617,-43.761
C04123=1014.196,-64.812,-112.890,-24.052,21.616,-43.756
C04124=1014.200,-64.404,-112.922,-24.053,21.615,-43.750
C04125=1014.204,-63.997,-112.955,-24.053,21.615,-43.744
C04126=1014.207,-63.590,-112.986,-24.054,21.615,-43.737
C04127=1014.212,-63.184,-113.019,-24.055,21.614,-43.732
C04128=1014.215,-62.778,-113.051,-24.056,21.613,-43.726
C04129=1014.219,-62.373,-113.083,-24.057,21.612,-43.720
C04130=1014.222,-61.968,-113.115,-24.057,21.611,-43.715
C04131=1014.226,-61.564,-113.146,-24.058,21.611,-43.708
C04132=1014.229,-61.159,-113.178,-24.059,21.610,-43.702
C04133=1014.233,-60.756,-113.210,-24.060,21.610,-43.697
C04134=1014.237,-60.354,-113.242,-24.061,21.610,-43.691
C04135=1014.240,-59.952,-113.273,-24.061,21.609,-43.686
C04136=1014.244,-59.551,-113.305,-24.062,21.608,-43.680
C04137=1014.247,-59.150,-113.337,-24.063,21.608,-43.673
C04138=1014.250,-58.750,-113.369,-24.064,21.607,-43.667
C04139=1014.254,-58.350,-113.400,-24.064,21.606,-43.662
C04140=1014.257,-57.951,-113.432,-24.065,21.606,-43.656
C04141=1014.260,-57.552,-113.463,-24.066,21.605,-43.651
C04142=1014.264,-57.154,-113.495,-24.067,21.604,-43.645
C04143=1014.267,-56.755,-113.526,-24.067,21.603,-43.639
C04144=1014.270,-56.358,-113.558,-24.068,21.603,-43.632
C04145=1014.273,-55.960,-113.589,-24.069,21.602,-43.627
C04146=1014.276,-55.562,-113.621,-24.070,21.603,-43.621
C04147=1014.279,-55.166,-113.653,-24.071,21.602,-43.616
C04148=1014.282,-54.768,-113.684,-24.071,21.601,-43.610
C04149=1014.285,-54.371,-113.715,-24.072,21.600,-43.604
C04150=1014.288,-53.974,-113.748,-24.073,21.599,-43.599
C04151=1014.290,-53.578,-113.779,-24.073,21.599,-43.593
C04152=1014.293,-53.180,-113.810,-24.074,21.598,-43.588
C04153=1014.296,-52.784,-113.842,-24.075,21.598,-43.581
C04154=1014.299,-52.386,-113.873,-24.076,21.598,-43.575
C04155=1014.302,-51.989,-113.905,-24.077,21.597,-43.570
C04156=1014.305,-51.593,-113.936,-24.077,21.596,-43.564
C04157=1014.307,-51.196,-113.968,-24.078,21.595,-43.558
C04158=1014.310,-50.799,-114.000,-24.079,21.595,-43.553
C04159=1014.313,-50.402,-114.032,-24.080,21.594,-43.547
C04160=1014.315,-50.004,-114.063,-24.080,21.593,-43.542
C04161=1014.317,-49.607,-114.095,-24.081,21.592,-43.536
C04162=1014.320,-49.211,-114.127,-24.082,21.592,-43.531
C04163=1014.323,-48.813,-114.158,-24.083,21.592,-43.525
C04164=1014.325,-48.416,-114.190,-24.084,21.592,-43.518
C04165=1014.328,-48.018,-114.221,-24.084,21.591,-43.512
C04166=1014.330,-47.622,-114.254,-24.085,21.590,-43.507
C04167=1014.333,-47.225,-114.285,-24.086,21.589,-43.501
C04168=1014.335,-46.827,-114.317,-24.086,21.588,-43.496
C04169=1014.338,-46.430,-114.348,-24.087,21.589,-43.490
C04170=1014.340,-46.033,-114.381,-24.088,21.588,-43.485
C04171=1014.341,-45.636,-114.413,-24.089,21.587,-43.479
C04172=1014.344,-45.238,-114.444,-24.089,21.586,-43.473
C04173=1014.346,-44.841,-114.476,-24.090,21.585,-43.468
C04174=1014.349,-44.443,-114.508,-24.091,21.585,-43.462
C04175=1014.350,-44.047,-114.540,-24.092,21.585,-43.457
C04176=1014.352,-43.649,-114.572,-24.092,21.584,-43.451
C04177=1014.355,-43.252,-114.604,-24.093,21.584,-43.444
C04178=1014.357,-42.854,-114.636,-24.094,21.583,-43.439
C04179=1014.359,-42.457,-114.667,-24.095,21.582,-43.433
C04180=1014.361,-42.060,-114.700,-24.096,21.582,-43.427
C04181=1014.363,-41.663,-114.732,-24.096,21.582,-43.422
C04182=1014.365,-41.266,-114.763,-24.097,21.581,-43.417
C04183=1014.367,-40.868,-114.795,-24.098,21.580,-43.411
C04184=1014.368,-40.470,-114.828,-24.099,21.579,-43.405
C04185=1014.370,-40.073,-114.859,-24.099,21.579,-43.400
C04186=1014.372,-39.676,-114.892,-24.100,21.578,-43.394
C04187=1014.375,-39.279,-114.924,-24.101,21.578,-43.389
C04188=1014.376,-38.882,-114.956,-24.102,21.577,-43.383
C04189=1014.378,-38.484,-114.988,-24.102,21.576,-43.378
C04190=1014.379,-38.086,-115.020,-24.103,21.576,-43.372
C04191=1014.381,-37.690,-115.052,-24.104,21.575,-43.366
C04192=1014.383,-37.292,-115.084,-24.105,21.575,-43.361
C04193=1014.385,-36.894,-115.117,-24.105,21.574,-43.356
C04194=1014.386,-36.497,-115.149,-24.106,21.573,-43.350
C04195=1014.388,-36.099,-115.181,-24.107,21.573,-43.344
C04196=1014.389,-35.702,-115.213,-24.107,21.572,-43.339
C04197=1014.391,-35.304,-115.245,-24.108,21.572,-43.334
C04198=1014.393,-34.907,-115.278,-24.109,21.571,-43.328
C04199=1014.394,-34.510,-115.310,-24.110,21.571,-43.321
C04200=1014.396,-34.113,-115.342,-24.111,21.570,-43.315
C04201=1014.397,-33.715,-115.374,-24.111,21.570,-43.310
C04202=1014.398,-33.317,-115.407,-24.112,21.570,-43.304
C04203=1014.399,-32.920,-115.438,-24.113,21.569,-43.299
C04204=1014.401,-32.523,-115.472,-24.114,21.568,-43.293
C04205=1014.402,-32.126,-115.504,-24.114,21.567,-43.287
C04206=1014.404,-31.728,-115.536,-24.115,21.568,-43.282
C04207=1014.405,-31.330,-115.568,-24.116,21.567,-43.277
C04208=1014.406,-30.933,-115.601,-24.117,21.566,-43.271
C04209=1014.408,-30.535,-115.633,-24.117,21.565,-43.265
C04210=1014.408,-30.138,-115.665,-24.118,21.565,-43.260
C04211=1014.410,-29.741,-115.699,-24.119,21.565,-43.255
C04212=1014.411,-29.343,-115.731,-24.120,21.564,-43.249
C04213=1014.412,-28.945,-115.763,-24.120,21.563,-43.243
C04214=1014.413,-28.548,-115.795,-24.121,21.562,-43.238
C04215=1014.414,-28.151,-115.828,-24.122,21.562,-43.232
C04216=1014.415,-27.753,-115.860,-24.123,21.562,-43.227
C04217=1014.416,-27.356,-115.893,-24.123,21.561,-43.221
C04218=1014.418,-26.958,-115.926,-24.124,21.560,-43.217
C04219=1014.418,-26.561,-115.958,-24.125,21.560,-43.212
C04220=1014.420,-26.163,-115.990,-24.125,21.559,-43.206
C04221=1014.420,-25.766,-116.023,-24.126,21.558,-43.201
C04222=1014.420,-25.368,-116.055,-24.127,21.558,-43.195
C04223=1014.422,-24.971,-116.089,-24.128,21.558,-43.190
C04224=1014.423,-24.574,-116.121,-24.128,21.557,-43.184
C04225=1014.424,-24.176,-116.154,-24.129,21.556,-43.178
C04226=1014.424,-23.778,-116.186,-24.130,21.556,-43.173
C04227=1014.425,-23.381,-116.218,-24.131,21.555,-43.168
C04228=1014.426,-22.983,-116.251,-24.131,21.555,-43.162
C04229=1014.427,-22.586,-116.284,-24.132,21.554,-43.156
C04230=1014.427,-22.189,-116.317,-24.133,21.554,-43.151
C04231=1014.428,-21.791,-116.350,-24.134,21.553,-43.146
C04232=1014.428,-21.393,-116.382,-24.134,21.552,-43.140
C04233=1014.430,-20.995,-116.415,-24.135,21.553,-43.135
C04234=1014.430,-20.598,-116.448,-24.136,21.552,-43.129
C04235=1014.430,-20.201,-116.481,-24.136,21.551,-43.123
C04236=1014.431,-19.789,-116.515,-24.138,21.551,-43.116
C04237=1014.431,-19.539,-116.535,-24.138,21.550,-43.113
C04238=1014.431,-19.252,-116.560,-24.139,21.550,-43.109
C04239=1014.432,-18.941,-116.585,-24.139,21.550,-43.107
C04240=1014.432,-18.629,-116.610,-24.139,21.549,-43.105
C04241=1014.433,-18.342,-116.635,-24.139,21.549,-43.101
C04242=1014.432,-18.093,-116.655,-24.140,21.548,-43.098
C04243=1014.433,-17.683,-116.688,-24.141,21.547,-43.090
C04244=1014.434,-17.285,-116.722,-24.142,21.548,-43.085
C04245=1014.434,-16.887,-116.754,-24.142,21.547,-43.079
C04246=1014.434,-16.488,-116.787,-24.143,21.546,-43.074
C04247=1014.434,-16.089,-116.821,-24.144,21.546,-43.068
C04248=1014.435,-15.688,-116.855,-24.145,21.545,-43.063
C04249=1014.435,-15.285,-116.888,-24.145,21.545,-43.057
C04250=1014.435,-14.879,-116.921,-24.146,21.544,-43.052
C04251=1014.435,-14.471,-116.955,-24.147,21.544,-43.046
C04252=1014.436,-14.059,-116.990,-24.148,21.543,-43.041
C04253=1014.436,-13.644,-117.024,-24.148,21.543,-43.035
C04254=1014.437,-13.227,-117.058,-24.149,21.542,-43.029
C04255=1014.436,-13.018,-117.076,-24.149,21.542,-43.028
C04256=1014.436,-12.596,-117.111,-24.150,21.541,-43.022
C04257=1014.436,-12.385,-117.129,-24.151,21.541,-43.019
C04258=1014.437,-12.174,-117.146,-24.151,21.540,-43.016
C04259=1014.436,-11.961,-117.164,-24.151,21.540,-43.013
C04260=1014.437,-11.749,-117.182,-24.152,21.540,-43.011
C04261=1014.437,-11.535,-117.199,-24.152,21.540,-43.007
C04262=1014.437,-11.321,-117.217,-24.152,21.539,-43.006
C04263=1014.436,-11.107,-117.235,-24.153,21.539,-43.002
C04264=1014.437,-10.893,-117.253,-24.153,21.539,-42.998
C04265=1014.436,-10.677,-117.271,-24.154,21.538,-42.996
C04266=1014.437,-10.463,-117.288,-24.154,21.539,-42.993
C04267=1014.436,-10.247,-117.307,-24.154,21.538,-42.991
C04268=1014.437,-10.030,-117.325,-24.155,21.538,-42.987
C04269=1014.436,-9.814,-117.343,-24.155,21.538,-42.985
C04270=1014.437,-9.598,-117.361,-24.156,21.537,-42.982
C04271=1014.436,-9.382,-117.379,-24.156,21.537,-42.980
C04272=1014.437,-9.166,-117.397,-24.156,21.536,-42.976
C04273=1014.436,-8.949,-117.416,-24.157,21.537,-42.973
C04274=1014.436,-8.732,-117.434,-24.157,21.536,-42.971
C04275=1014.436,-8.516,-117.452,-24.158,21.536,-42.967
C04276=1014.436,-8.299,-117.470,-24.158,21.536,-42.965
C04277=1014.436,-8.081,-117.488,-24.158,21.535,-42.961
C04278=1014.435,-7.864,-117.507,-24.159,21.535,-42.959
C04279=1014.436,-7.644,-117.524,-24.159,21.534,-42.956
C04280=1014.436,-7.424,-117.542,-24.160,21.535,-42.952
C04281=1014.436,-7.202,-117.561,-24.160,21.534,-42.950
C04282=1014.435,-6.980,-117.580,-24.160,21.534,-42.947
C04283=1014.435,-6.756,-117.599,-24.161,21.533,-42.944
C04284=1014.435,-6.532,-117.618,-24.161,21.533,-42.941
C04285=1014.435,-6.309,-117.637,-24.161,21.533,-42.939
C04286=1014.435,-6.084,-117.656,-24.162,21.533,-42.935
C04287=1014.434,-5.860,-117.674,-24.162,21.532,-42.934
C04288=1014.434,-5.636,-117.693,-24.163,21.532,-42.930
C04289=1014.434,-5.414,-117.711,-24.163,21.532,-42.927
C04290=1014.434,-5.193,-117.729,-24.163,21.532,-42.925
C04291=1014.434,-4.973,-117.749,-24.164,21.531,-42.921
C04292=1014.434,-4.754,-117.767,-24.164,21.531,-42.919
C04293=1014.433,-4.538,-117.784,-24.165,21.531,-42.915
C04294=1014.433,-4.322,-117.803,-24.165,21.530,-42.913
C04295=1014.434,-4.109,-117.821,-24.165,21.530,-42.910
C04296=1014.433,-3.897,-117.839,-24.166,21.530,-42.908
C04297=1014.432,-3.685,-117.856,-24.166,21.530,-42.904
C04298=1014.433,-3.263,-117.892,-24.167,21.529,-42.899
C04299=1014.432,-2.844,-117.927,-24.168,21.529,-42.893
C04300=1014.431,-2.428,-117.963,-24.169,21.529,-42.888
C04301=1014.431,-2.012,-117.997,-24.169,21.528,-42.882
C04302=1014.430,-1.600,-118.033,-24.170,21.527,-42.877
C04303=1014.429,-1.190,-118.067,-24.171,21.527,-42.872
C04304=1014.429,-0.782,-118.102,-24.171,21.526,-42.867
C04305=1014.428,-0.376,-118.136,-24.172,21.525,-42.862
C04306=1014.427,0.028,-118.169,-24.173,21.525,-42.857
C04307=1014.427,0.429,-118.203,-24.173,21.525,-42.851
C04308=1014.427,0.830,-118.237,-24.174,21.525,-42.846
C04309=1014.425,1.228,-118.271,-24.175,21.523,-42.841
C04310=1014.425,1.626,-118.305,-24.175,21.524,-42.836
C04311=1014.425,2.012,-118.337,-24.176,21.523,-42.833
C04312=1014.423,2.364,-118.367,-24.177,21.522,-42.827
C04313=1014.423,2.687,-118.395,-24.177,21.522,-42.823
C04314=1014.422,3.000,-118.421,-24.178,21.521,-42.817
C04315=1014.421,3.328,-118.449,-24.179,21.521,-42.812
C04316=1014.421,3.688,-118.479,-24.179,21.521,-42.809
C04317=1014.420,4.077,-118.512,-24.180,21.520,-42.805
C04318=1014.419,4.473,-118.545,-24.180,21.519,-42.799
C04319=1014.418,4.868,-118.579,-24.181,21.520,-42.794
C04320=1014.418,5.263,-118.613,-24.182,21.519,-42.790
C04321=1014.416,5.657,-118.646,-24.182,21.518,-42.785
C04322=1014.416,6.051,-118.680,-24.183,21.519,-42.779
C04323=1014.415,6.444,-118.714,-24.184,21.517,-42.775
C04324=1014.413,6.837,-118.747,-24.185,21.517,-42.770
C04325=1014.412,7.227,-118.779,-24.185,21.517,-42.764
C04326=1014.412,7.615,-118.813,-24.186,21.516,-42.761
C04327=1014.410,7.999,-118.846,-24.187,21.516,-42.755
C04328=1014.410,8.380,-118.878,-24.187,21.515,-42.751
C04329=1014.408,8.758,-118.910,-24.188,21.515,-42.746
C04330=1014.407,9.134,-118.943,-24.189,21.514,-42.740
C04331=1014.406,9.510,-118.974,-24.189,21.514,-42.737
C04332=1014.405,9.886,-119.006,-24.190,21.513,-42.731
C04333=1014.404,10.265,-119.039,-24.191,21.513,-42.726
C04334=1014.403,10.645,-119.071,-24.191,21.513,-42.722
C04335=1014.402,11.028,-119.104,-24.192,21.512,-42.716
C04336=1014.400,11.414,-119.137,-24.192,21.511,-42.713
C04337=1014.399,11.800,-119.170,-24.193,21.512,-42.707
C04338=1014.397,12.186,-119.203,-24.193,21.510,-42.703
C04339=1014.397,12.573,-119.236,-24.194,21.510,-42.698
C04340=1014.395,12.960,-119.269,-24.195,21.511,-42.693
C04341=1014.394,13.346,-119.302,-24.196,21.509,-42.689
C04342=1014.392,13.734,-119.335,-24.196,21.509,-42.683
C04343=1014.391,14.121,-119.368,-24.197,21.509,-42.680
C04344=1014.389,14.510,-119.402,-24.198,21.508,-42.674
C04345=1014.388,14.899,-119.435,-24.198,21.508,-42.670
C04346=1014.387,15.288,-119.468,-24.199,21.507,-42.665
C04347=1014.386,15.678,-119.502,-24.200,21.507,-42.659
C04348=1014.383,16.069,-119.535,-24.200,21.506,-42.656
C04349=1014.382,16.461,-119.570,-24.201,21.506,-42.650
C04350=1014.381,16.854,-119.603,-24.201,21.505,-42.646
C04351=1014.379,17.247,-119.637,-24.202,21.505,-42.641
C04352=1014.378,17.641,-119.671,-24.203,21.505,-42.635
C04353=1014.376,18.036,-119.705,-24.203,21.504,-42.632
C04354=1014.374,18.432,-119.739,-24.204,21.503,-42.626
C04355=1014.372,18.829,-119.773,-24.205,21.503,-42.622
C04356=1014.372,19.027,-119.790,-24.205,21.503,-42.619
C04357=1014.370,19.437,-119.825,-24.206,21.503,-42.613
C04358=1014.369,19.673,-119.845,-24.206,21.502,-42.610
C04359=1014.368,19.938,-119.869,-24.207,21.503,-42.606
C04360=1014.367,20.226,-119.894,-24.207,21.501,-42.604
C04361=1014.365,20.523,-119.919,-24.207,21.501,-42.602
C04362=1014.363,20.814,-119.944,-24.208,21.502,-42.599
C04363=1014.362,21.086,-119.968,-24.208,21.501,-42.597
C04364=1014.362,21.331,-119.989,-24.209,21.501,-42.593
C04365=1014.359,21.744,-120.024,-24.210,21.501,-42.586
C04366=1014.358,22.119,-120.057,-24.210,21.500,-42.584
C04367=1014.356,22.442,-120.085,-24.211,21.500,-42.580
C04368=1014.355,22.706,-120.108,-24.211,21.500,-42.577
C04369=1014.354,22.939,-120.128,-24.211,21.499,-42.573
C04370=1014.353,23.174,-120.148,-24.212,21.498,-42.567
C04371=1014.351,23.445,-120.172,-24.213,21.498,-42.564
C04372=1014.350,23.775,-120.200,-24.213,21.498,-42.562
C04373=1014.348,24.158,-120.233,-24.213,21.497,-42.558
C04374=1014.346,24.558,-120.268,-24.214,21.497,-42.553
C04375=1014.344,24.958,-120.302,-24.215,21.497,-42.549
C04376=1014.342,25.356,-120.337,-24.215,21.496,-42.543
C04377=1014.340,25.755,-120.372,-24.216,21.496,-42.540
C04378=1014.337,26.155,-120.406,-24.217,21.496,-42.534
C04379=1014.335,26.554,-120.441,-24.218,21.495,-42.529
C04380=1014.333,26.954,-120.475,-24.218,21.494,-42.525
C04381=1014.331,27.352,-120.510,-24.219,21.495,-42.520
C04382=1014.329,27.752,-120.544,-24.219,21.493,-42.516
C04383=1014.327,28.152,-120.580,-24.220,21.493,-42.510
C04384=1014.324,28.551,-120.614,-24.221,21.493,-42.507
C04385=1014.322,28.951,-120.649,-24.221,21.492,-42.501
C04386=1014.320,29.350,-120.683,-24.222,21.492,-42.497
C04387=1014.318,29.750,-120.719,-24.223,21.492,-42.492
C04388=1014.315,30.149,-120.753,-24.223,21.491,-42.488
C04389=1014.313,30.549,-120.788,-24.224,21.491,-42.483
C04390=1014.311,30.948,-120.822,-24.224,21.490,-42.479
C04391=1014.308,31.347,-120.858,-24.225,21.490,-42.474
C04392=1014.306,31.747,-120.892,-24.226,21.489,-42.469
C04393=1014.304,32.147,-120.927,-24.226,21.489,-42.464
C04394=1014.301,32.547,-120.962,-24.227,21.489,-42.461
C04395=1014.298,32.946,-120.997,-24.228,21.489,-42.455
C04396=1014.296,33.346,-121.032,-24.228,21.487,-42.451
C04397=1014.294,33.746,-121.066,-24.229,21.488,-42.446
C04398=1014.291,34.145,-121.101,-24.229,21.487,-42.442
C04399=1014.288,34.545,-121.136,-24.230,21.486,-42.437
C04400=1014.286,34.945,-121.171,-24.231,21.486,-42.433
C04401=1014.283,35.345,-121.206,-24.231,21.486,-42.428
C04402=1014.280,35.744,-121.241,-24.232,21.486,-42.424
C04403=1014.277,36.144,-121.276,-24.233,21.485,-42.418
C04404=1014.275,36.544,-121.311,-24.233,21.484,-42.414
C04405=1014.273,36.944,-121.346,-24.234,21.485,-42.409
C04406=1014.269,37.343,-121.381,-24.235,21.484,-42.405
C04407=1014.267,37.743,-121.415,-24.235,21.483,-42.400
C04408=1014.264,38.143,-121.451,-24.236,21.483,-42.396
C04409=1014.262,38.543,-121.486,-24.237,21.483,-42.391
C04410=1014.258,38.943,-121.521,-24.237,21.483,-42.387
C04411=1014.255,39.342,-121.556,-24.238,21.482,-42.383
C04412=1014.253,39.742,-121.591,-24.238,21.481,-42.378
C04413=1014.250,40.142,-121.626,-24.239,21.481,-42.374
C04414=1014.246,40.542,-121.662,-24.240,21.481,-42.369
C04415=1014.244,40.942,-121.697,-24.240,21.481,-42.365
C04416=1014.241,41.342,-121.731,-24.241,21.480,-42.359
C04417=1014.237,41.742,-121.766,-24.241,21.479,-42.356
C04418=1014.235,42.141,-121.802,-24.242,21.479,-42.352
C04419=1014.232,42.542,-121.837,-24.243,21.479,-42.347
C04420=1014.229,42.942,-121.872,-24.243,21.479,-42.343
C04421=1014.226,43.341,-121.907,-24.244,21.479,-42.338
C04422=1014.222,43.742,-121.942,-24.244,21.477,-42.333
C04423=1014.219,44.142,-121.978,-24.245,21.477,-42.330
C04424=1014.216,44.541,-122.013,-24.246,21.477,-42.325
C04425=1014.213,44.942,-122.048,-24.246,21.477,-42.321
C04426=1014.210,45.342,-122.083,-24.247,21.477,-42.316
C04427=1014.207,45.742,-122.119,-24.247,21.475,-42.311
C04428=1014.203,46.141,-122.154,-24.248,21.475,-42.308
C04429=1014.200,46.541,-122.189,-24.249,21.475,-42.302
C04430=1014.197,46.942,-122.224,-24.249,21.475,-42.299
C04431=1014.193,47.342,-122.259,-24.250,21.474,-42.295
C04432=1014.190,47.742,-122.295,-24.251,21.474,-42.290
C04433=1014.187,48.142,-122.330,-24.251,21.474,-42.286
C04434=1014.183,48.541,-122.365,-24.251,21.472,-42.282
C04435=1014.180,48.942,-122.401,-24.252,21.473,-42.277
C04436=1014.177,49.342,-122.436,-24.253,21.472,-42.273
C04437=1014.173,49.742,-122.471,-24.254,21.472,-42.268
C04438=1014.169,50.142,-122.507,-24.254,21.472,-42.264
C04439=1014.166,50.542,-122.542,-24.255,21.471,-42.260
C04440=1014.162,50.942,-122.578,-24.255,21.471,-42.255
C04441=1014.159,51.343,-122.613,-24.256,21.471,-42.251
C04442=1014.155,51.742,-122.648,-24.256,21.470,-42.247
C04443=1014.151,52.143,-122.683,-24.257,21.469,-42.243
C04444=1014.147,52.543,-122.718,-24.258,21.469,-42.238
C04445=1014.144,52.943,-122.755,-24.258,21.469,-42.234
C04446=1014.140,53.342,-122.790,-24.259,21.468,-42.230
C04447=1014.137,53.743,-122.825,-24.259,21.468,-42.225
C04448=1014.132,54.143,-122.861,-24.260,21.468,-42.221
C04449=1014.129,54.543,-122.896,-24.260,21.468,-42.218
C04450=1014.125,54.943,-122.931,-24.261,21.468,-42.212
C04451=1014.122,55.344,-122.966,-24.262,21.467,-42.209
C04452=1014.117,55.744,-123.002,-24.262,21.467,-42.205
C04453=1014.114,56.144,-123.038,-24.263,21.465,-42.201
C04454=1014.110,56.543,-123.073,-24.264,21.466,-42.196
C04455=1014.106,56.944,-123.109,-24.264,21.465,-42.192
C04456=1014.102,57.344,-123.144,-24.264,21.465,-42.188
C04457=1014.098,57.744,-123.180,-24.265,21.465,-42.183
C04458=1014.094,58.144,-123.215,-24.266,21.464,-42.179
C04459=1014.090,58.544,-123.250,-24.266,21.464,-42.175
C04460=1014.086,58.945,-123.286,-24.267,21.463,-42.172
C04461=1014.082,59.345,-123.321,-24.268,21.464,-42.166
C04462=1014.077,59.744,-123.358,-24.268,21.463,-42.163
C04463=1014.074,60.145,-123.393,-24.269,21.463,-42.159
C04464=1014.069,60.545,-123.429,-24.269,21.462,-42.155
C04465=1014.065,60.944,-123.464,-24.270,21.462,-42.150
C04466=1014.061,61.345,-123.500,-24.270,21.462,-42.146
C04467=1014.057,61.745,-123.535,-24.271,21.461,-42.142
C04468=1014.052,62.145,-123.571,-24.271,21.461,-42.139
C04469=1014.048,62.565,-123.608,-24.272,21.460,-42.133
C04470=1014.046,62.818,-123.630,-24.272,21.460,-42.131
C04471=1014.043,63.085,-123.654,-24.273,21.460,-42.129
C04472=1014.040,63.335,-123.676,-24.273,21.459,-42.127
C04473=1014.038,63.553,-123.696,-24.274,21.460,-42.124
C04474=1014.035,63.759,-123.714,-24.274,21.460,-42.122
C04475=1014.033,63.977,-123.734,-24.274,21.459,-42.120
C04476=1014.030,64.206,-123.754,-24.274,21.459,-42.116
C04477=1014.028,64.442,-123.775,-24.275,21.459,-42.115
C04478=1014.025,64.678,-123.796,-24.275,21.458,-42.113
C04479=1014.022,64.908,-123.817,-24.275,21.458,-42.111
C04480=1014.020,65.129,-123.836,-24.276,21.459,-42.108
C04481=1014.017,65.342,-123.856,-24.276,21.458,-42.106
C04482=1014.013,65.750,-123.891,-24.277,21.458,-42.102
C04483=1014.009,66.147,-123.927,-24.277,21.457,-42.098
C04484=1014.004,66.549,-123.963,-24.278,21.457,-42.094
C04485=1014.000,66.951,-123.998,-24.278,21.457,-42.089
C04486=1013.995,67.354,-124.034,-24.279,21.457,-42.085
C04487=1013.990,67.758,-124.070,-24.279,21.456,-42.082
C04488=1013.986,68.165,-124.107,-24.280,21.456,-42.078
C04489=1013.980,68.572,-124.143,-24.280,21.455,-42.074
C04490=1013.976,68.980,-124.179,-24.281,21.455,-42.069
C04491=1013.971,69.391,-124.216,-24.282,21.455,-42.065
C04492=1013.966,69.802,-124.253,-24.282,21.454,-42.061
C04493=1013.961,70.213,-124.290,-24.283,21.454,-42.058
C04494=1013.956,70.624,-124.326,-24.283,21.453,-42.054
C04495=1013.951,71.034,-124.363,-24.284,21.454,-42.049
C04496=1013.946,71.446,-124.399,-24.285,21.453,-42.045
C04497=1013.941,71.858,-124.436,-24.285,21.453,-42.041
C04498=1013.936,72.271,-124.473,-24.285,21.452,-42.037
C04499=1013.931,72.686,-124.510,-24.286,21.452,-42.034
C04500=1013.925,73.104,-124.547,-24.287,21.452,-42.028
C04501=1013.920,73.524,-124.585,-24.287,21.452,-42.025
C04502=1013.918,73.736,-124.604,-24.288,21.451,-42.023
C04503=1013.915,73.947,-124.623,-24.288,21.451,-42.021
C04504=1013.911,74.160,-124.642,-24.288,21.451,-42.019
C04505=1013.909,74.373,-124.660,-24.288,21.451,-42.017
C04506=1013.907,74.587,-124.680,-24.289,21.450,-42.015
C04507=1013.904,74.800,-124.699,-24.289,21.451,-42.012
C04508=1013.901,75.013,-124.718,-24.289,21.451,-42.010
C04509=1013.898,75.226,-124.737,-24.290,21.450,-42.008
C04510=1013.893,75.646,-124.775,-24.290,21.450,-42.004
C04511=1013.887,76.057,-124.811,-24.291,21.449,-42.001
C04512=1013.882,76.459,-124.847,-24.291,21.449,-41.997
C04513=1013.877,76.854,-124.882,-24.292,21.449,-41.994
C04514=1013.872,77.242,-124.917,-24.292,21.448,-41.989
C04515=1013.866,77.628,-124.952,-24.293,21.447,-41.986
C04516=1013.861,78.015,-124.986,-24.293,21.448,-41.980
C04517=1013.856,78.405,-125.021,-24.294,21.447,-41.977
C04518=1013.851,78.802,-125.056,-24.294,21.447,-41.973
C04519=1013.845,79.207,-125.093,-24.295,21.447,-41.970
C04520=1013.842,79.414,-125.111,-24.295,21.447,-41.968
C04521=1013.837,79.832,-125.149,-24.296,21.446,-41.964
C04522=1013.834,80.044,-125.167,-24.296,21.446,-41.962
C04523=1013.830,80.256,-125.187,-24.296,21.446,-41.960
C04524=1013.828,80.469,-125.206,-24.297,21.446,-41.958
C04525=1013.825,80.682,-125.225,-24.297,21.445,-41.956
C04526=1013.821,80.895,-125.244,-24.297,21.445,-41.955
C04527=1013.819,81.106,-125.263,-24.297,21.445,-41.953
C04528=1013.816,81.319,-125.282,-24.298,21.445,-41.951
C04529=1013.813,81.531,-125.301,-24.298,21.445,-41.949
C04530=1013.809,81.742,-125.320,-24.298,21.444,-41.947
C04531=1013.807,81.954,-125.339,-24.299,21.445,-41.944
C04532=1013.803,82.165,-125.358,-24.299,21.444,-41.942
C04533=1013.798,82.586,-125.396,-24.299,21.444,-41.938
C04534=1013.792,83.007,-125.433,-24.300,21.444,-41.935
C04535=1013.786,83.425,-125.470,-24.300,21.444,-41.931
C04536=1013.779,83.843,-125.508,-24.301,21.443,-41.927
C04537=1013.773,84.258,-125.545,-24.301,21.443,-41.923
C04538=1013.767,84.672,-125.582,-24.302,21.443,-41.920
C04539=1013.762,85.084,-125.619,-24.302,21.442,-41.916
C04540=1013.756,85.495,-125.656,-24.303,21.442,-41.912
C04541=1013.749,85.904,-125.692,-24.303,21.441,-41.908
C04542=1013.743,86.311,-125.729,-24.304,21.442,-41.905
C04543=1013.737,86.716,-125.765,-24.304,21.441,-41.901
C04544=1013.735,86.869,-125.779,-24.305,21.441,-41.899
C04545=1013.716,88.066,-125.886,-24.412,21.838,-41.648
C04546=1013.713,88.290,-125.906,-24.431,21.913,-41.601
C04547=1013.710,88.513,-125.926,-24.451,21.987,-41.554
C04548=1013.706,88.738,-125.946,-24.471,22.063,-41.508
C04549=1013.702,88.965,-125.966,-24.491,22.139,-41.461
C04550=1013.699,89.195,-125.987,-24.511,22.217,-41.412
C04551=1013.695,89.427,-126.008,-24.531,22.295,-41.364
C04552=1013.692,89.664,-126.029,-24.553,22.376,-41.314
C04553=1013.687,89.947,-126.054,-24.578,22.473,-41.254
C04554=1013.682,90.280,-126.084,-24.607,22.586,-41.186
C04555=1013.676,90.599,-126.112,-24.634,22.695,-41.119
C04556=1013.673,90.859,-126.135,-24.657,22.785,-41.064
C04557=1013.669,91.094,-126.156,-24.677,22.866,-41.016
C04558=1013.666,91.329,-126.178,-24.698,22.947,-40.966
C04559=1013.662,91.564,-126.199,-24.718,23.029,-40.919
C04560=1013.658,91.799,-126.219,-24.739,23.110,-40.869
C04561=1013.654,92.034,-126.241,-24.759,23.193,-40.820
C04562=1013.651,92.269,-126.261,-24.780,23.275,-40.770
C04563=1013.647,92.505,-126.282,-24.800,23.358,-40.723
C04564=1013.644,92.740,-126.304,-24.820,23.440,-40.674
C04565=1013.639,92.975,-126.324,-24.840,23.523,-40.625
C04566=1013.635,93.210,-126.345,-24.860,23.606,-40.577
C04567=1013.632,93.445,-126.367,-24.881,23.690,-40.527
C04568=1013.628,93.680,-126.387,-24.901,23.774,-40.478
C04569=1013.624,93.916,-126.409,-24.921,23.857,-40.430
C04570=1013.621,94.150,-126.429,-24.941,23.941,-40.382
C04571=1013.616,94.385,-126.451,-24.961,24.026,-40.333
C04572=1013.613,94.621,-126.471,-24.981,24.109,-40.284
C04573=1013.609,94.856,-126.493,-25.001,24.194,-40.235
C04574=1013.605,95.090,-126.513,-25.021,24.279,-40.188
C04575=1013.601,95.326,-126.534,-25.041,24.364,-40.139
C04576=1013.598,95.561,-126.555,-25.060,24.450,-40.090
C04577=1013.593,95.796,-126.576,-25.080,24.534,-40.043
C04578=1013.590,96.031,-126.597,-25.100,24.621,-39.994
C04579=1013.586,96.266,-126.619,-25.119,24.706,-39.946
C04580=1013.583,96.501,-126.639,-25.139,24.792,-39.898
C04581=1013.578,96.736,-126.660,-25.159,24.879,-39.849
C04582=1013.575,96.971,-126.681,-25.178,24.965,-39.801
C04583=1013.571,97.207,-126.702,-25.198,25.052,-39.753
C04584=1013.567,97.441,-126.722,-25.218,25.140,-39.705
C04585=1013.563,97.677,-126.744,-25.237,25.226,-39.657
C04586=1013.560,97.911,-126.765,-25.256,25.314,-39.609
C04587=1013.555,98.146,-126.786,-25.276,25.402,-39.561
C04588=1013.552,98.382,-126.806,-25.295,25.489,-39.514
C04589=1013.548,98.616,-126.828,-25.314,25.578,-39.465
C04590=1013.544,98.851,-126.848,-25.333,25.665,-39.418
C04591=1013.540,99.087,-126.869,-25.353,25.754,-39.370
C04592=1013.536,99.322,-126.889,-25.372,25.844,-39.322
C04593=1013.532,99.557,-126.911,-25.391,25.931,-39.275
C04594=1013.529,99.792,-126.932,-25.410,26.020,-39.227
C04595=1013.524,100.027,-126.953,-25.429,26.110,-39.180
C04596=1013.521,100.261,-126.974,-25.448,26.200,-39.133
C04597=1013.516,100.496,-126.995,-25.467,26.289,-39.085
C04598=1013.513,100.732,-127.015,-25.486,26.380,-39.038
C04599=1013.508,100.967,-127.036,-25.505,26.470,-38.989
C04600=1013.505,101.202,-127.058,-25.524,26.560,-38.942
C04601=1013.501,101.437,-127.078,-25.542,26.651,-38.895
C04602=1013.497,101.672,-127.099,-25.561,26.741,-38.849
C04603=1013.493,101.907,-127.120,-25.580,26.833,-38.801
C04604=1013.489,102.141,-127.141,-25.598,26.924,-38.754
C04605=1013.485,102.377,-127.162,-25.617,27.016,-38.707
C04606=1013.481,102.612,-127.182,-25.636,27.106,-38.660
C04607=1013.477,102.847,-127.203,-25.654,27.198,-38.613
C04608=1013.471,103.241,-127.238,-25.685,27.353,-38.534
C04609=1013.465,103.551,-127.266,-25.709,27.475,-38.473
C04610=1013.462,103.787,-127.286,-25.728,27.569,-38.426
C04611=1013.457,104.021,-127.308,-25.746,27.661,-38.379
C04612=1013.453,104.257,-127.329,-25.764,27.754,-38.333
C04613=1013.449,104.491,-127.349,-25.782,27.847,-38.286
C04614=1013.445,104.727,-127.370,-25.801,27.941,-38.240
C04615=1013.441,104.961,-127.391,-25.819,28.036,-38.193
C04616=1013.437,105.197,-127.412,-25.837,28.129,-38.146
C04617=1013.433,105.431,-127.432,-25.855,28.223,-38.101
C04618=1013.429,105.667,-127.453,-25.873,28.318,-38.055
C04619=1013.425,105.901,-127.474,-25.891,28.413,-38.008
C04620=1013.421,106.136,-127.495,-25.908,28.507,-37.963
C04621=1013.417,106.371,-127.516,-25.926,28.602,-37.916
C04622=1013.413,106.607,-127.537,-25.944,28.698,-37.871
C04623=1013.409,106.842,-127.557,-25.962,28.793,-37.824
C04624=1013.405,107.076,-127.578,-25.980,28.889,-37.778
C04625=1013.401,107.311,-127.599,-25.997,28.984,-37.734
C04626=1013.397,107.546,-127.620,-26.015,29.080,-37.688
C04627=1013.393,107.781,-127.641,-26.032,29.177,-37.642
C04628=1013.389,108.016,-127.661,-26.050,29.273,-37.596
C04629=1013.384,108.251,-127.682,-26.067,29.370,-37.551
C04630=1013.381,108.486,-127.702,-26.084,29.467,-37.505
C04631=1013.376,108.721,-127.724,-26.102,29.564,-37.460
C04632=1013.373,108.956,-127.744,-26.119,29.661,-37.415
C04633=1013.368,109.191,-127.765,-26.136,29.759,-37.370
C04634=1013.364,109.426,-127.786,-26.154,29.857,-37.324
C04635=1013.360,109.661,-127.806,-26.171,29.955,-37.279
C04636=1013.356,109.896,-127.827,-26.188,30.052,-37.234
C04637=1013.352,110.131,-127.848,-26.205,30.151,-37.189
C04638=1013.348,110.366,-127.869,-26.222,30.249,-37.145
C04639=1013.344,110.600,-127.889,-26.239,30.348,-37.099
C04640=1013.340,110.836,-127.910,-26.255,30.447,-37.055
C04641=1013.336,111.070,-127.931,-26.272,30.547,-37.010
C04642=1013.331,111.305,-127.951,-26.289,30.645,-36.966
C04643=1013.327,111.541,-127.972,-26.306,30.745,-36.922
C04644=1013.323,111.776,-127.993,-26.322,30.845,-36.877
C04645=1013.319,112.011,-128.014,-26.339,30.945,-36.832
C04646=1013.315,112.245,-128.035,-26.356,31.045,-36.788
C04647=1013.311,112.480,-128.055,-26.372,31.145,-36.744
C04648=1013.307,112.715,-128.076,-26.389,31.246,-36.700
C04649=1013.302,112.950,-128.097,-26.405,31.347,-36.656
C04650=1013.298,113.185,-128.117,-26.421,31.447,-36.612
C04651=1013.294,113.420,-128.138,-26.438,31.549,-36.569
C04652=1013.290,113.655,-128.158,-26.454,31.650,-36.525
C04653=1013.286,113.890,-128.179,-26.470,31.751,-36.482
C04654=1013.282,114.126,-128.200,-26.486,31.853,-36.437
C04655=1013.278,114.360,-128.220,-26.502,31.955,-36.394
C04656=1013.273,114.595,-128.241,-26.518,32.057,-36.351
C04657=1013.269,114.830,-128.261,-26.534,32.160,-36.307
C04658=1013.265,115.065,-128.282,-26.550,32.262,-36.264
C04659=1013.261,115.300,-128.302,-26.566,32.365,-36.221
C04660=1013.256,115.535,-128.323,-26.582,32.469,-36.177
C04661=1013.253,115.770,-128.344,-26.598,32.571,-36.135
C04662=1013.248,116.005,-128.365,-26.614,32.675,-36.092
C04663=1013.244,116.239,-128.385,-26.629,32.779,-36.049
C04664=1013.240,116.475,-128.407,-26.645,32.883,-36.005
C04665=1013.236,116.710,-128.427,-26.661,32.987,-35.962
C04666=1013.232,116.944,-128.447,-26.676,33.090,-35.921
C04667=1013.227,117.179,-128.468,-26.691,33.195,-35.879
C04668=1013.224,117.415,-128.489,-26.707,33.299,-35.836
C04669=1013.218,117.700,-128.514,-26.726,33.427,-35.784
C04670=1013.211,118.120,-128.551,-26.753,33.615,-35.709
C04671=1013.207,118.354,-128.571,-26.768,33.720,-35.667
C04672=1013.202,118.589,-128.592,-26.783,33.825,-35.625
C04673=1013.198,118.824,-128.612,-26.798,33.931,-35.582
C04674=1013.194,119.059,-128.633,-26.813,34.037,-35.541
C04675=1013.190,119.295,-128.652,-26.828,34.143,-35.500
C04676=1013.185,119.530,-128.673,-26.843,34.250,-35.458
C04677=1013.182,119.765,-128.694,-26.858,34.356,-35.417
C04678=1013.177,120.000,-128.715,-26.873,34.463,-35.375
C04679=1013.172,120.235,-128.735,-26.888,34.570,-35.333
C04680=1013.168,120.469,-128.755,-26.902,34.677,-35.293
C04681=1013.164,120.705,-128.777,-26.917,34.781,-35.253
C04682=1013.161,120.939,-128.798,-26.930,34.879,-35.215
C04683=1013.157,121.174,-128.818,-26.943,34.977,-35.177
C04684=1013.153,121.409,-128.839,-26.957,35.076,-35.139
C04685=1013.149,121.644,-128.859,-26.970,35.175,-35.102
C04686=1013.145,121.879,-128.880,-26.983,35.274,-35.065
C04687=1013.142,122.114,-128.901,-26.996,35.372,-35.027
C04688=1013.137,122.349,-128.922,-27.009,35.472,-34.990
C04689=1013.133,122.584,-128.943,-27.022,35.571,-34.954
C04690=1013.129,122.819,-128.963,-27.035,35.670,-34.917
C04691=1013.125,123.055,-128.984,-27.048,35.770,-34.880
C04692=1013.121,123.289,-129.005,-27.061,35.869,-34.844
C04693=1013.118,123.524,-129.026,-27.074,35.969,-34.807
C04694=1013.114,123.759,-129.046,-27.087,36.070,-34.770
C04695=1013.110,123.994,-129.067,-27.100,36.170,-34.734
C04696=1013.106,124.229,-129.087,-27.113,36.271,-34.696
C04697=1013.101,124.465,-129.109,-27.125,36.371,-34.661
C04698=1013.098,124.699,-129.129,-27.138,36.472,-34.625
C04699=1013.094,124.934,-129.151,-27.150,36.573,-34.588
C04700=1013.090,125.169,-129.171,-27.163,36.673,-34.553
C04701=1013.086,125.404,-129.192,-27.175,36.775,-34.516
C04702=1013.082,125.639,-129.212,-27.188,36.877,-34.480
C04703=1013.078,125.874,-129.233,-27.200,36.977,-34.444
C04704=1013.074,126.109,-129.253,-27.213,37.079,-34.408
C04705=1013.071,126.344,-129.275,-27.225,37.182,-34.372
C04706=1013.066,126.579,-129.295,-27.238,37.284,-34.336
C04707=1013.063,126.814,-129.316,-27.250,37.385,-34.302
C04708=1013.058,127.049,-129.337,-27.262,37.487,-34.266
C04709=1013.054,127.284,-129.357,-27.274,37.590,-34.231
C04710=1013.050,127.519,-129.378,-27.286,37.693,-34.195
C04711=1013.046,127.755,-129.398,-27.298,37.796,-34.160
C04712=1013.043,127.990,-129.419,-27.310,37.899,-34.125
C04713=1013.038,128.225,-129.440,-27.322,38.002,-34.090
C04714=1013.035,128.460,-129.460,-27.334,38.105,-34.056
C04715=1013.031,128.695,-129.482,-27.346,38.208,-34.021
C04716=1013.027,128.930,-129.502,-27.358,38.312,-33.987
C04717=1013.022,129.165,-129.523,-27.370,38.416,-33.952
C04718=1013.019,129.400,-129.544,-27.382,38.520,-33.917
C04719=1013.014,129.635,-129.564,-27.394,38.624,-33.882
C04720=1013.011,129.870,-129.585,-27.405,38.728,-33.849
C04721=1013.007,130.105,-129.605,-27.417,38.833,-33.813
C04722=1013.003,130.341,-129.626,-27.429,38.937,-33.780
C04723=1012.999,130.575,-129.646,-27.440,39.042,-33.747
C04724=1012.995,130.811,-129.668,-27.452,39.146,-33.712
C04725=1012.991,131.045,-129.688,-27.463,39.251,-33.679
C04726=1012.986,131.340,-129.713,-27.478,39.383,-33.635
C04727=1012.980,131.751,-129.750,-27.497,39.567,-33.577
C04728=1012.975,131.986,-129.770,-27.509,39.673,-33.543
C04729=1012.971,132.221,-129.791,-27.520,39.778,-33.511
C04730=1012.967,132.456,-129.812,-27.531,39.885,-33.478
C04731=1012.963,132.691,-129.832,-27.543,39.990,-33.444
C04732=1012.959,132.926,-129.852,-27.554,40.097,-33.411
C04733=1012.955,133.162,-129.873,-27.565,40.204,-33.378
C04734=1012.951,133.396,-129.894,-27.576,40.309,-33.345
C04735=1012.947,133.632,-129.915,-27.587,40.416,-33.313
C04736=1012.943,133.866,-129.935,-27.598,40.523,-33.280
C04737=1012.940,134.102,-129.955,-27.609,40.630,-33.248
C04738=1012.936,134.337,-129.977,-27.620,40.737,-33.215
C04739=1012.931,134.577,-129.997,-27.631,40.846,-33.182
C04740=1012.927,134.872,-130.023,-27.645,40.980,-33.142
C04741=1012.921,135.157,-130.048,-27.658,41.111,-33.103
C04742=1012.918,135.390,-130.068,-27.668,41.218,-33.071
C04743=1012.914,135.615,-130.088,-27.679,41.322,-33.040
C04744=1012.907,136.034,-130.124,-27.697,41.513,-32.984
C04745=1012.900,136.420,-130.158,-27.715,41.692,-32.932
C04746=1012.894,136.803,-130.192,-27.732,41.868,-32.881
C04747=1012.887,137.219,-130.227,-27.751,42.061,-32.826
C04748=1012.881,137.603,-130.262,-27.768,42.239,-32.775
C04749=1012.874,138.023,-130.298,-27.786,42.434,-32.720
C04750=1012.869,138.276,-130.320,-27.797,42.552,-32.687
C04751=1012.865,138.549,-130.344,-27.809,42.679,-32.652
C04752=1012.860,138.844,-130.369,-27.822,42.816,-32.613
C04753=1012.855,139.151,-130.396,-27.835,42.960,-32.574
C04754=1012.850,139.464,-130.423,-27.848,43.106,-32.534
C04755=1012.845,139.772,-130.450,-27.862,43.251,-32.495
C04756=1012.840,140.068,-130.476,-27.874,43.390,-32.458
C04757=1012.834,140.342,-130.499,-27.886,43.520,-32.422
C04758=1012.830,140.594,-130.522,-27.897,43.639,-32.390
C04759=1012.826,140.887,-130.548,-27.909,43.777,-32.353
C04760=1012.822,141.143,-130.570,-27.920,43.897,-32.323
C04761=1012.818,141.353,-130.588,-27.928,43.997,-32.297
C04762=1012.814,141.598,-130.609,-27.939,44.114,-32.266
C04763=1012.810,141.837,-130.630,-27.948,44.226,-32.236
C04764=1012.807,142.077,-130.650,-27.958,44.340,-32.207
C04765=1012.802,142.315,-130.671,-27.968,44.454,-32.178
C04766=1012.798,142.555,-130.692,-27.978,44.568,-32.149
C04767=1012.795,142.795,-130.713,-27.988,44.682,-32.119
C04768=1012.791,143.035,-130.734,-27.998,44.797,-32.091
C04769=1012.787,143.275,-130.755,-28.007,44.912,-32.062
C04770=1012.782,143.515,-130.775,-28.017,45.027,-32.034
C04771=1012.778,143.756,-130.796,-28.027,45.142,-32.004
C04772=1012.775,143.997,-130.817,-28.037,45.258,-31.976
C04773=1012.769,144.326,-130.846,-28.050,45.416,-31.937
C04774=1012.762,144.720,-130.880,-28.066,45.606,-31.890
C04775=1012.759,144.962,-130.901,-28.075,45.722,-31.863
C04776=1012.755,145.204,-130.922,-28.085,45.839,-31.835
C04777=1012.750,145.445,-130.943,-28.094,45.956,-31.807
C04778=1012.746,145.688,-130.964,-28.104,46.072,-31.779
C04779=1012.743,145.929,-130.984,-28.113,46.189,-31.751
C04780=1012.739,146.171,-131.005,-28.123,46.306,-31.724
C04781=1012.735,146.414,-131.027,-28.132,46.425,-31.696
C04782=1012.731,146.656,-131.047,-28.142,46.542,-31.669
C04783=1012.727,146.899,-131.068,-28.151,46.661,-31.642
C04784=1012.723,147.147,-131.090,-28.161,46.782,-31.614
C04785=1012.719,147.402,-131.112,-28.171,46.906,-31.586
C04786=1012.715,147.663,-131.135,-28.181,47.033,-31.557
C04787=1012.710,147.934,-131.157,-28.191,47.166,-31.527
C04788=1012.706,148.211,-131.182,-28.202,47.302,-31.497
C04789=1012.701,148.497,-131.207,-28.212,47.442,-31.465
C04790=1012.697,148.788,-131.232,-28.224,47.585,-31.435
C04791=1012.691,149.084,-131.258,-28.235,47.730,-31.403
C04792=1012.687,149.384,-131.283,-28.246,47.878,-31.372
C04793=1012.682,149.683,-131.309,-28.258,48.026,-31.340
C04794=1012.677,149.983,-131.335,-28.269,48.174,-31.309
C04795=1012.672,150.280,-131.360,-28.280,48.321,-31.278
C04796=1012.668,150.572,-131.385,-28.291,48.465,-31.248
C04797=1012.663,150.858,-131.410,-28.301,48.606,-31.218
C04798=1012.659,151.137,-131.434,-28.312,48.745,-31.190
C04799=1012.654,151.408,-131.457,-28.322,48.879,-31.163
C04800=1012.649,151.671,-131.480,-28.332,49.009,-31.136
C04801=1012.646,151.925,-131.502,-28.341,49.137,-31.110
C04802=1012.642,152.174,-131.524,-28.350,49.259,-31.086
C04803=1012.638,152.418,-131.545,-28.359,49.381,-31.062
C04804=1012.634,152.660,-131.565,-28.368,49.501,-31.038
C04805=1012.630,152.901,-131.586,-28.377,49.622,-31.013
C04806=1012.627,153.143,-131.607,-28.385,49.743,-30.991
C04807=1012.623,153.385,-131.628,-28.394,49.863,-30.967
C04808=1012.619,153.626,-131.648,-28.403,49.984,-30.945
C04809=1012.616,153.867,-131.669,-28.412,50.104,-30.922
C04810=1012.612,154.108,-131.690,-28.421,50.225,-30.899
C04811=1012.608,154.348,-131.710,-28.429,50.345,-30.877
C04812=1012.604,154.590,-131.731,-28.438,50.466,-30.854
C04813=1012.600,154.830,-131.751,-28.447,50.587,-30.833
C04814=1012.596,155.069,-131.772,-28.455,50.707,-30.810
C04815=1012.592,155.309,-131.793,-28.464,50.828,-30.788
C04816=1012.588,155.549,-131.813,-28.473,50.949,-30.767
C04817=1012.585,155.788,-131.834,-28.481,51.069,-30.747
C04818=1012.581,156.028,-131.855,-28.490,51.189,-30.725
C04819=1012.578,156.267,-131.875,-28.498,51.310,-30.703
C04820=1012.574,156.507,-131.896,-28.507,51.430,-30.682
C04821=1012.571,156.768,-131.918,-28.516,51.562,-30.660
C04822=1012.566,156.985,-131.937,-28.524,51.672,-30.640
C04823=1012.563,157.225,-131.957,-28.533,51.792,-30.621
C04824=1012.560,157.463,-131.978,-28.541,51.914,-30.601
C04825=1012.556,157.701,-131.998,-28.550,52.033,-30.580
C04826=1012.552,157.937,-132.018,-28.558,52.153,-30.561
C04827=1012.549,158.174,-132.039,-28.567,52.273,-30.542
C04828=1012.545,158.410,-132.058,-28.575,52.393,-30.521
C04829=1012.541,158.645,-132.079,-28.584,52.513,-30.502
C04830=1012.538,158.880,-132.099,-28.592,52.632,-30.483
C04831=1012.534,159.116,-132.119,-28.600,52.752,-30.465
C04832=1012.531,159.353,-132.139,-28.609,52.871,-30.446
C04833=1012.527,159.587,-132.159,-28.617,52.990,-30.427
C04834=1012.524,159.820,-132.180,-28.626,53.108,-30.410
C04835=1012.521,160.051,-132.201,-28.630,53.171,-30.399
C04836=1012.520,160.285,-132.225,-28.631,53.181,-30.398
C04837=1012.520,160.526,-132.250,-28.631,53.192,-30.394
C04838=1012.518,160.775,-132.276,-28.632,53.203,-30.393
C04839=1012.518,161.038,-132.304,-28.632,53.216,-30.390
C04840=1012.517,161.315,-132.332,-28.633,53.228,-30.388
C04841=1012.516,161.608,-132.362,-28.634,53.241,-30.384
C04842=1012.514,161.912,-132.394,-28.635,53.253,-30.382
C04843=1012.513,162.217,-132.425,-28.635,53.267,-30.379
C04844=1012.512,162.509,-132.456,-28.636,53.280,-30.376
C04845=1012.510,162.817,-132.487,-28.637,53.294,-30.373
C04846=1012.509,163.111,-132.518,-28.638,53.306,-30.371
C04847=1012.509,163.374,-132.545,-28.638,53.318,-30.369
C04848=1012.508,163.611,-132.570,-28.639,53.329,-30.366
C04849=1012.507,163.832,-132.592,-28.640,53.339,-30.364
C04850=1012.506,164.053,-132.616,-28.640,53.348,-30.361
C04851=1012.504,164.441,-132.656,-28.641,53.366,-30.358
C04852=1012.503,164.759,-132.690,-28.642,53.380,-30.356
C04853=1012.502,165.061,-132.721,-28.643,53.393,-30.354
C04854=1012.501,165.297,-132.745,-28.643,53.403,-30.351
C04855=1012.500,165.532,-132.770,-28.644,53.414,-30.349
C04856=1012.499,165.768,-132.794,-28.645,53.424,-30.347
C04857=1012.498,166.003,-132.818,-28.645,53.434,-30.345
C04858=1012.497,166.239,-132.843,-28.646,53.445,-30.342
C04859=1012.497,166.474,-132.868,-28.646,53.455,-30.340
C04860=1012.496,166.710,-132.892,-28.647,53.465,-30.339
C04861=1012.495,166.946,-132.917,-28.647,53.476,-30.335
C04862=1012.494,167.181,-132.941,-28.648,53.486,-30.334
C04863=1012.493,167.416,-132.966,-28.649,53.497,-30.331
C04864=1012.492,167.652,-132.990,-28.649,53.507,-30.330
C04865=1012.491,167.887,-133.015,-28.650,53.519,-30.327
C04866=1012.490,168.123,-133.039,-28.651,53.529,-30.325
C04867=1012.490,168.359,-133.064,-28.651,53.539,-30.324
C04868=1012.489,168.595,-133.089,-28.652,53.549,-30.322
C04869=1012.488,168.830,-133.114,-28.652,53.560,-30.319
C04870=1012.487,169.066,-133.137,-28.653,53.570,-30.317
C04871=1012.486,169.301,-133.163,-28.654,53.581,-30.316
C04872=1012.485,169.537,-133.187,-28.654,53.592,-30.313
C04873=1012.485,169.772,-133.212,-28.655,53.603,-30.312
C04874=1012.484,170.008,-133.236,-28.656,53.614,-30.309
C04875=1012.482,170.243,-133.261,-28.656,53.626,-30.306
C04876=1012.482,170.479,-133.285,-28.657,53.636,-30.304
C04877=1012.481,170.714,-133.310,-28.658,53.646,-30.303
C04878=1012.480,170.951,-133.335,-28.658,53.656,-30.301
C04879=1012.480,171.186,-133.359,-28.659,53.667,-30.298
C04880=1012.478,171.422,-133.384,-28.660,53.678,-30.297
C04881=1012.477,171.657,-133.409,-28.660,53.688,-30.295
C04882=1012.477,171.893,-133.433,-28.661,53.699,-30.293
C04883=1012.476,172.128,-133.458,-28.662,53.711,-30.290
C04884=1012.475,172.364,-133.482,-28.662,53.721,-30.289
C04885=1012.474,172.599,-133.507,-28.663,53.733,-30.286
C04886=1012.474,172.836,-133.532,-28.664,53.743,-30.284
C04887=1012.472,173.071,-133.557,-28.664,53.753,-30.283
C04888=1012.471,173.307,-133.581,-28.665,53.763,-30.281
C04889=1012.471,173.542,-133.606,-28.666,53.775,-30.279
C04890=1012.470,173.778,-133.631,-28.666,53.785,-30.277
C04891=1012.469,174.014,-133.655,-28.667,53.796,-30.274
C04892=1012.469,174.249,-133.680,-28.668,53.807,-30.273
C04893=1012.468,174.485,-133.705,-28.668,53.818,-30.270
C04894=1012.467,174.721,-133.730,-28.669,53.830,-30.268
C04895=1012.465,174.956,-133.754,-28.670,53.841,-30.267
C04896=1012.466,175.192,-133.779,-28.670,53.851,-30.265
C04897=1012.464,175.428,-133.803,-28.671,53.862,-30.262
C04898=1012.463,175.663,-133.828,-28.672,53.872,-30.260
C04899=1012.463,175.899,-133.854,-28.672,53.883,-30.259
C04900=1012.462,176.135,-133.878,-28.673,53.894,-30.256
C04901=1012.461,176.370,-133.903,-28.674,53.905,-30.255
C04902=1012.460,176.607,-133.928,-28.674,53.916,-30.253
C04903=1012.459,176.842,-133.953,-28.675,53.928,-30.250
C04904=1012.458,177.077,-133.976,-28.676,53.939,-30.250
C04905=1012.458,177.313,-134.002,-28.677,53.951,-30.247
C04906=1012.457,177.549,-134.027,-28.677,53.961,-30.245
C04907=1012.456,177.785,-134.052,-28.678,53.971,-30.244
C04908=1012.455,178.021,-134.077,-28.679,53.982,-30.241
C04909=1012.455,178.256,-134.101,-28.679,53.992,-30.240
C04910=1012.454,178.492,-134.126,-28.680,54.004,-30.237
C04911=1012.453,178.727,-134.151,-28.681,54.015,-30.236
C04912=1012.452,178.964,-134.176,-28.681,54.026,-30.233
C04913=1012.452,179.199,-134.200,-28.682,54.038,-30.232
C04914=1012.451,179.435,-134.226,-28.683,54.049,-30.231
C04915=1012.450,179.671,-134.250,-28.683,54.060,-30.227
C04916=1012.449,179.907,-134.276,-28.684,54.071,-30.227
C04917=1012.448,180.142,-134.301,-28.685,54.081,-30.225
C04918=1012.448,180.378,-134.325,-28.686,54.093,-30.222
C04919=1012.447,180.614,-134.350,-28.686,54.103,-30.221
C04920=1012.446,180.849,-134.374,-28.687,54.115,-30.218
C04921=1012.445,181.085,-134.400,-28.688,54.126,-30.217
C04922=1012.444,181.321,-134.425,-28.688,54.137,-30.215
C04923=1012.443,181.557,-134.450,-28.689,54.149,-30.213
C04924=1012.443,181.792,-134.474,-28.690,54.161,-30.210
C04925=1012.443,182.028,-134.500,-28.691,54.172,-30.209
C04926=1012.442,182.265,-134.524,-28.691,54.182,-30.208
C04927=1012.441,182.500,-134.549,-28.692,54.193,-30.205
C04928=1012.440,182.736,-134.575,-28.693,54.204,-30.204
C04929=1012.439,182.972,-134.599,-28.693,54.215,-30.201
C04930=1012.439,183.207,-134.624,-28.694,54.226,-30.200
C04931=1012.438,183.443,-134.649,-28.695,54.238,-30.198
C04932=1012.437,183.679,-134.674,-28.695,54.249,-30.196
C04933=1012.436,183.915,-134.699,-28.697,54.261,-30.196
C04934=1012.436,184.151,-134.725,-28.697,54.273,-30.193
C04935=1012.435,184.386,-134.750,-28.698,54.285,-30.191
C04936=1012.434,184.622,-134.774,-28.699,54.295,-30.189
C04937=1012.434,184.858,-134.799,-28.699,54.305,-30.188
C04938=1012.433,185.093,-134.824,-28.700,54.316,-30.185
C04939=1012.432,185.330,-134.849,-28.701,54.327,-30.184
C04940=1012.432,185.566,-134.875,-28.701,54.339,-30.182
C04941=1012.431,185.801,-134.900,-28.702,54.351,-30.179
C04942=1012.430,186.037,-134.925,-28.703,54.362,-30.179
C04943=1012.429,186.273,-134.949,-28.704,54.374,-30.177
C04944=1012.428,186.509,-134.975,-28.705,54.387,-30.175
C04945=1012.429,186.745,-135.000,-28.705,54.397,-30.174
C04946=1012.428,186.980,-135.025,-28.706,54.408,-30.171
C04947=1012.427,187.216,-135.050,-28.707,54.419,-30.171
C04948=1012.426,187.452,-135.075,-28.707,54.430,-30.167
C04949=1012.425,187.688,-135.100,-28.708,54.441,-30.166
C04950=1012.425,187.924,-135.126,-28.709,54.453,-30.164
C04951=1012.424,188.160,-135.150,-28.710,54.464,-30.164
C04952=1012.423,188.395,-135.175,-28.711,54.476,-30.162
C04953=1012.423,188.631,-135.201,-28.712,54.489,-30.160
C04954=1012.422,188.867,-135.226,-28.712,54.500,-30.158
C04955=1012.422,189.102,-135.251,-28.713,54.511,-30.157
C04956=1012.421,189.339,-135.276,-28.714,54.522,-30.154
C04957=1012.420,189.575,-135.301,-28.714,54.533,-30.153
C04958=1012.419,189.810,-135.326,-28.715,54.545,-30.151
C04959=1012.419,190.046,-135.352,-28.716,54.556,-30.150
C04960=1012.418,190.282,-135.377,-28.717,54.567,-30.147
C04961=1012.418,190.519,-135.402,-28.718,54.580,-30.146
C04962=1012.417,190.754,-135.427,-28.718,54.591,-30.145
C04963=1012.416,190.990,-135.452,-28.719,54.603,-30.143
C04964=1012.416,191.226,-135.478,-28.720,54.615,-30.141
C04965=1012.415,191.462,-135.503,-28.721,54.627,-30.139
C04966=1012.414,191.697,-135.528,-28.722,54.638,-30.138
C04967=1012.413,191.934,-135.553,-28.722,54.648,-30.137
C04968=1012.414,192.169,-135.578,-28.723,54.660,-30.135
C04969=1012.413,192.405,-135.603,-28.724,54.671,-30.134
C04970=1012.413,192.641,-135.629,-28.725,54.683,-30.132
C04971=1012.412,192.877,-135.654,-28.726,54.695,-30.130
C04972=1012.411,193.113,-135.679,-28.726,54.707,-30.128
C04973=1012.411,193.348,-135.705,-28.727,54.720,-30.126
C04974=1012.410,193.584,-135.730,-28.728,54.732,-30.125
C04975=1012.409,193.820,-135.755,-28.729,54.742,-30.123
C04976=1012.408,194.056,-135.780,-28.730,54.753,-30.122
C04977=1012.408,194.292,-135.806,-28.730,54.765,-30.120
C04978=1012.407,194.528,-135.831,-28.731,54.776,-30.119
C04979=1012.407,194.764,-135.857,-28.732,54.788,-30.117
C04980=1012.406,195.000,-135.882,-28.733,54.800,-30.115
C04981=1012.406,195.236,-135.907,-28.734,54.812,-30.114
C04982=1012.405,195.471,-135.933,-28.735,54.823,-30.113
C04983=1012.404,195.707,-135.958,-28.735,54.836,-30.111
C04984=1012.404,195.943,-135.983,-28.736,54.848,-30.110
C04985=1012.403,196.179,-136.009,-28.737,54.860,-30.107
C04986=1012.403,196.415,-136.034,-28.738,54.871,-30.107
C04987=1012.402,196.651,-136.060,-28.739,54.882,-30.106
C04988=1012.402,196.887,-136.085,-28.739,54.893,-30.103
C04989=1012.401,197.122,-136.110,-28.740,54.905,-30.101
C04990=1012.400,197.358,-136.136,-28.741,54.917,-30.101
C04991=1012.400,197.594,-136.161,-28.742,54.929,-30.100
C04992=1012.399,197.830,-136.187,-28.743,54.941,-30.097
C04993=1012.400,198.066,-136.212,-28.744,54.954,-30.096
C04994=1012.398,198.314,-136.238,-28.745,54.966,-30.094
C04995=1012.398,198.705,-136.281,-28.746,54.986,-30.091
C04996=1012.397,199.096,-136.322,-28.748,55.006,-30.090
C04997=1012.396,199.337,-136.348,-28.748,55.018,-30.088
C04998=1012.396,199.567,-136.373,-28.749,55.030,-30.086
C04999=1012.396,199.799,-136.398,-28.750,55.041,-30.085
C05000=1012.396,200.041,-136.424,-28.751,55.054,-30.084
C05001=1012.395,200.294,-136.452,-28.752,55.066,-30.082
C05002=1012.394,200.549,-136.480,-28.753,55.079,-30.081
C05003=1012.393,200.788,-136.505,-28.754,55.091,-30.079
C05004=1012.393,201.012,-136.529,-28.754,55.103,-30.077
C05005=1012.393,201.227,-136.552,-28.755,55.114,-30.076
C05006=1012.392,201.440,-136.575,-28.756,55.124,-30.075
C05007=1012.391,201.850,-136.620,-28.757,55.145,-30.072
C05008=1012.391,202.068,-136.644,-28.758,55.156,-30.071
C05009=1012.394,203.312,-136.781,-28.910,55.091,-30.750
C05010=1012.397,203.559,-136.808,-28.911,55.104,-30.749
C05011=1012.398,203.803,-136.834,-28.912,55.115,-30.748
C05012=1012.399,204.047,-136.861,-28.913,55.127,-30.747
C05013=1012.401,204.292,-136.887,-28.914,55.139,-30.747
C05014=1012.403,204.537,-136.914,-28.915,55.150,-30.747
C05015=1012.404,204.780,-136.941,-28.917,55.161,-30.746
C05016=1012.407,205.025,-136.967,-28.918,55.174,-30.745
C05017=1012.408,205.268,-136.994,-28.919,55.185,-30.745
C05018=1012.410,205.512,-137.020,-28.920,55.196,-30.744
C05019=1012.412,205.756,-137.047,-28.921,55.209,-30.743
C05020=1012.414,205.999,-137.073,-28.922,55.220,-30.743
C05021=1012.416,206.242,-137.100,-28.923,55.231,-30.742
C05022=1012.416,206.486,-137.126,-28.925,55.243,-30.742
C05023=1012.418,206.729,-137.152,-28.926,55.255,-30.741
C05024=1012.421,206.971,-137.180,-28.927,55.266,-30.740
C05025=1012.422,207.214,-137.206,-28.928,55.278,-30.740
C05026=1012.424,207.457,-137.232,-28.929,55.289,-30.738
C05027=1012.426,207.700,-137.259,-28.930,55.301,-30.738
C05028=1012.428,207.942,-137.285,-28.931,55.312,-30.737
C05029=1012.430,208.184,-137.312,-28.932,55.323,-30.737
C05030=1012.432,208.428,-137.338,-28.933,55.334,-30.737
C05031=1012.433,208.669,-137.365,-28.934,55.347,-30.735
C05032=1012.435,208.912,-137.391,-28.935,55.358,-30.735
C05033=1012.437,209.154,-137.418,-28.937,55.369,-30.735
C05034=1012.439,209.397,-137.444,-28.938,55.381,-30.733
C05035=1012.441,209.639,-137.471,-28.939,55.393,-30.733
C05036=1012.442,209.882,-137.498,-28.940,55.403,-30.732
C05037=1012.444,210.123,-137.524,-28.941,55.415,-30.732
C05038=1012.446,210.367,-137.551,-28.942,55.426,-30.731
C05039=1012.448,210.608,-137.578,-28.943,55.438,-30.730
C05040=1012.450,210.852,-137.604,-28.944,55.449,-30.729
C05041=1012.452,211.094,-137.630,-28.946,55.461,-30.729
C05042=1012.454,211.337,-137.657,-28.947,55.472,-30.729
C05043=1012.456,211.580,-137.684,-28.948,55.484,-30.727
C05044=1012.458,211.823,-137.710,-28.949,55.495,-30.727
C05045=1012.459,212.066,-137.737,-28.950,55.507,-30.727
C05046=1012.462,212.309,-137.765,-28.951,55.517,-30.726
C05047=1012.464,212.552,-137.791,-28.952,55.529,-30.726
C05048=1012.466,212.795,-137.818,-28.953,55.540,-30.725
C05049=1012.467,213.039,-137.845,-28.954,55.552,-30.724
C05050=1012.469,213.283,-137.871,-28.955,55.563,-30.723
C05051=1012.471,213.527,-137.898,-28.957,55.575,-30.723
C05052=1012.473,213.771,-137.925,-28.958,55.586,-30.723
C05053=1012.475,214.015,-137.951,-28.959,55.597,-30.723
C05054=1012.477,214.259,-137.979,-28.960,55.608,-30.722
C05055=1012.479,214.505,-138.006,-28.961,55.621,-30.721
C05056=1012.481,214.749,-138.033,-28.962,55.631,-30.720
C05057=1012.483,214.995,-138.060,-28.964,55.643,-30.720
C05058=1012.485,215.239,-138.087,-28.965,55.654,-30.720
C05059=1012.487,215.485,-138.114,-28.966,55.666,-30.720
C05060=1012.489,215.730,-138.141,-28.967,55.676,-30.719
C05061=1012.492,215.976,-138.168,-28.968,55.688,-30.719
C05062=1012.494,216.221,-138.196,-28.969,55.699,-30.718
C05063=1012.496,216.467,-138.223,-28.970,55.711,-30.717
C05064=1012.497,216.716,-138.250,-28.971,55.722,-30.716
C05065=1012.500,216.970,-138.278,-28.973,55.735,-30.715
C05066=1012.502,217.230,-138.308,-28.973,55.746,-30.713
C05067=1012.504,217.495,-138.336,-28.974,55.759,-30.712
C05068=1012.507,217.775,-138.367,-28.976,55.772,-30.711
C05069=1012.509,218.064,-138.400,-28.977,55.785,-30.712
C05070=1012.512,218.357,-138.433,-28.979,55.799,-30.713
C05071=1012.514,218.653,-138.465,-28.981,55.811,-30.714
C05072=1012.517,218.957,-138.498,-28.982,55.825,-30.714
C05073=1012.519,219.253,-138.531,-28.984,55.838,-30.715
C05074=1012.521,219.534,-138.563,-28.985,55.851,-30.714
C05075=1012.524,219.807,-138.593,-28.986,55.863,-30.713
C05076=1012.527,220.067,-138.621,-28.987,55.876,-30.712
C05077=1012.529,220.316,-138.649,-28.988,55.888,-30.710
C05078=1012.531,220.561,-138.677,-28.989,55.898,-30.709
C05079=1012.534,220.807,-138.704,-28.990,55.909,-30.708
C05080=1012.535,221.053,-138.732,-28.992,55.921,-30.709
C05081=1012.538,221.299,-138.759,-28.993,55.932,-30.708
C05082=1012.540,221.544,-138.787,-28.994,55.943,-30.707
C05083=1012.542,221.790,-138.814,-28.995,55.953,-30.707
C05084=1012.544,222.035,-138.841,-28.996,55.963,-30.707
C05085=1012.547,222.282,-138.869,-28.997,55.973,-30.706
C05086=1012.549,222.527,-138.896,-28.998,55.984,-30.705
C05087=1012.551,222.772,-138.924,-28.999,55.996,-30.705
C05088=1012.554,223.019,-138.951,-29.000,56.007,-30.705
C05089=1012.556,223.264,-138.979,-29.002,56.018,-30.705
C05090=1012.558,223.510,-139.006,-29.002,56.030,-30.703
C05091=1012.560,223.755,-139.033,-29.004,56.041,-30.703
C05092=1012.563,224.002,-139.060,-29.005,56.054,-30.702
C05093=1012.565,224.247,-139.088,-29.006,56.065,-30.701
C05094=1012.567,224.492,-139.116,-29.007,56.075,-30.702
C05095=1012.570,224.739,-139.143,-29.008,56.086,-30.701
C05096=1012.572,224.984,-139.170,-29.009,56.096,-30.700
C05097=1012.574,225.229,-139.198,-29.010,56.107,-30.700
C05098=1012.577,225.475,-139.226,-29.011,56.118,-30.699
C05099=1012.579,225.721,-139.253,-29.012,56.129,-30.699
C05100=1012.581,225.966,-139.281,-29.014,56.140,-30.699
C05101=1012.584,226.212,-139.309,-29.015,56.151,-30.698
C05102=1012.586,226.458,-139.336,-29.016,56.164,-30.697
C05103=1012.588,226.703,-139.363,-29.017,56.175,-30.697
C05104=1012.591,226.949,-139.392,-29.018,56.186,-30.697
C05105=1012.593,227.195,-139.419,-29.019,56.195,-30.697
C05106=1012.595,227.439,-139.446,-29.020,56.206,-30.696
C05107=1012.598,227.686,-139.474,-29.021,56.217,-30.696
C05108=1012.600,227.931,-139.501,-29.023,56.227,-30.696
C05109=1012.602,228.176,-139.529,-29.024,56.238,-30.696
C05110=1012.605,228.423,-139.557,-29.024,56.249,-30.694
C05111=1012.607,228.668,-139.585,-29.026,56.261,-30.694
C05112=1012.610,228.914,-139.612,-29.027,56.272,-30.693
C05113=1012.612,229.159,-139.639,-29.028,56.284,-30.692
C05114=1012.614,229.404,-139.668,-29.029,56.296,-30.692
C05115=1012.617,229.651,-139.695,-29.031,56.306,-30.693
C05116=1012.620,229.896,-139.723,-29.031,56.316,-30.692
C05117=1012.622,230.142,-139.750,-29.033,56.326,-30.693
C05118=1012.625,230.387,-139.778,-29.033,56.336,-30.691
C05119=1012.626,230.633,-139.806,-29.035,56.347,-30.691
C05120=1012.629,230.878,-139.834,-29.036,56.357,-30.690
C05121=1012.632,231.124,-139.861,-29.037,56.369,-30.690
C05122=1012.635,231.369,-139.889,-29.038,56.380,-30.690
C05123=1012.637,231.614,-139.917,-29.039,56.392,-30.688
C05124=1012.639,231.861,-139.945,-29.040,56.404,-30.689
C05125=1012.642,232.106,-139.973,-29.042,56.415,-30.688
C05126=1012.645,232.352,-140.000,-29.043,56.424,-30.688
C05127=1012.647,232.597,-140.028,-29.044,56.435,-30.687
C05128=1012.650,232.842,-140.056,-29.044,56.445,-30.686
C05129=1012.653,233.088,-140.083,-29.046,56.455,-30.687
C05130=1012.654,233.333,-140.112,-29.047,56.465,-30.686
C05131=1012.657,233.579,-140.140,-29.048,56.476,-30.686
C05132=1012.660,233.824,-140.167,-29.049,56.487,-30.685
C05133=1012.663,234.070,-140.195,-29.050,56.499,-30.685
C05134=1012.665,234.315,-140.223,-29.051,56.511,-30.684
C05135=1012.667,234.561,-140.251,-29.052,56.522,-30.684
C05136=1012.670,234.806,-140.279,-29.053,56.533,-30.683
C05137=1012.673,235.052,-140.307,-29.055,56.542,-30.683
C05138=1012.675,235.297,-140.335,-29.056,56.553,-30.683
C05139=1012.678,235.543,-140.362,-29.057,56.562,-30.683
C05140=1012.681,235.789,-140.391,-29.058,56.573,-30.682
C05141=1012.683,236.034,-140.419,-29.059,56.583,-30.681
C05142=1012.686,236.279,-140.447,-29.060,56.594,-30.681
C05143=1012.689,236.524,-140.475,-29.061,56.605,-30.680
C05144=1012.692,236.770,-140.502,-29.062,56.617,-30.681
C05145=1012.694,237.015,-140.530,-29.064,56.628,-30.681
C05146=1012.696,237.261,-140.559,-29.064,56.640,-30.679
C05147=1012.699,237.506,-140.587,-29.066,56.650,-30.680
C05148=1012.702,237.752,-140.615,-29.067,56.660,-30.678
C05149=1012.705,237.997,-140.643,-29.068,56.669,-30.678
C05150=1012.708,238.242,-140.671,-29.068,56.679,-30.677
C05151=1012.711,238.488,-140.699,-29.070,56.689,-30.678
C05152=1012.713,238.733,-140.727,-29.071,56.700,-30.677
C05153=1012.715,238.979,-140.755,-29.072,56.710,-30.677
C05154=1012.719,239.225,-140.783,-29.073,56.721,-30.676
C05155=1012.721,239.470,-140.811,-29.074,56.733,-30.677
C05156=1012.724,239.715,-140.839,-29.075,56.744,-30.675
C05157=1012.726,239.960,-140.867,-29.076,56.756,-30.675
C05158=1012.729,240.206,-140.895,-29.078,56.765,-30.675
C05159=1012.732,240.452,-140.924,-29.078,56.775,-30.674
C05160=1012.735,240.696,-140.951,-29.079,56.784,-30.674
C05161=1012.738,240.942,-140.980,-29.080,56.795,-30.673
C05162=1012.741,241.187,-141.008,-29.081,56.804,-30.673
C05163=1012.743,241.432,-141.037,-29.083,56.815,-30.673
C05164=1012.746,241.678,-141.065,-29.084,56.826,-30.672
C05165=1012.749,241.923,-141.093,-29.085,56.837,-30.672
C05166=1012.752,242.168,-141.121,-29.086,56.848,-30.672
C05167=1012.755,242.414,-141.149,-29.087,56.861,-30.671
C05168=1012.758,242.659,-141.177,-29.088,56.872,-30.670
C05169=1012.760,242.905,-141.206,-29.089,56.880,-30.670
C05170=1012.763,243.150,-141.234,-29.090,56.889,-30.670
C05171=1012.766,243.395,-141.263,-29.091,56.900,-30.669
C05172=1012.769,243.641,-141.291,-29.092,56.909,-30.669
C05173=1012.772,243.886,-141.319,-29.093,56.920,-30.669
C05174=1012.774,244.132,-141.348,-29.094,56.930,-30.668
C05175=1012.777,244.377,-141.376,-29.095,56.941,-30.668
C05176=1012.780,244.622,-141.404,-29.097,56.952,-30.667
C05177=1012.783,244.867,-141.432,-29.098,56.963,-30.667
C05178=1012.786,245.113,-141.461,-29.099,56.974,-30.667
C05179=1012.790,245.358,-141.489,-29.100,56.984,-30.666
C05180=1012.792,245.603,-141.518,-29.101,56.994,-30.666
C05181=1012.795,245.848,-141.546,-29.102,57.003,-30.666
C05182=1012.798,246.094,-141.574,-29.103,57.013,-30.664
C05183=1012.801,246.339,-141.603,-29.104,57.023,-30.665
C05184=1012.804,246.585,-141.631,-29.105,57.033,-30.664
C05185=1012.806,246.830,-141.660,-29.106,57.043,-30.664
C05186=1012.810,247.075,-141.688,-29.107,57.054,-30.663
C05187=1012.813,247.320,-141.717,-29.108,57.065,-30.663
C05188=1012.816,247.566,-141.745,-29.109,57.077,-30.663
C05189=1012.819,247.810,-141.773,-29.110,57.088,-30.661
C05190=1012.822,248.056,-141.802,-29.111,57.097,-30.661
C05191=1012.824,248.301,-141.831,-29.112,57.107,-30.661
C05192=1012.828,248.547,-141.859,-29.113,57.116,-30.661
C05193=1012.831,248.792,-141.888,-29.114,57.126,-30.660
C05194=1012.834,249.037,-141.916,-29.115,57.135,-30.660
C05195=1012.838,249.282,-141.945,-29.116,57.146,-30.660
C05196=1012.839,249.528,-141.973,-29.117,57.156,-30.659
C05197=1012.843,249.772,-142.002,-29.119,57.167,-30.659
C05198=1012.846,250.018,-142.031,-29.120,57.178,-30.658
C05199=1012.849,250.263,-142.059,-29.121,57.189,-30.658
C05200=1012.852,250.509,-142.088,-29.122,57.201,-30.657
C05201=1012.856,250.754,-142.116,-29.123,57.209,-30.656
C05202=1012.858,251.000,-142.145,-29.124,57.219,-30.656
C05203=1012.862,251.245,-142.174,-29.125,57.228,-30.656
C05204=1012.864,251.489,-142.203,-29.126,57.237,-30.656
C05205=1012.868,251.734,-142.231,-29.127,57.247,-30.655
C05206=1012.871,251.979,-142.260,-29.128,57.258,-30.654
C05207=1012.874,252.225,-142.289,-29.128,57.268,-30.653
C05208=1012.877,252.470,-142.317,-29.130,57.278,-30.653
C05209=1012.880,252.715,-142.346,-29.131,57.290,-30.653
C05210=1012.884,252.960,-142.375,-29.132,57.301,-30.653
C05211=1012.887,253.206,-142.403,-29.133,57.312,-30.652
C05212=1012.889,253.451,-142.433,-29.134,57.320,-30.651
C05213=1012.893,253.696,-142.462,-29.135,57.329,-30.652
C05214=1012.896,253.941,-142.491,-29.136,57.338,-30.652
C05215=1012.899,254.187,-142.519,-29.137,57.348,-30.650
C05216=1012.903,254.432,-142.548,-29.138,57.357,-30.651
C05217=1012.905,254.677,-142.577,-29.139,57.368,-30.650
C05218=1012.909,254.922,-142.606,-29.140,57.378,-30.649
C05219=1012.912,255.167,-142.635,-29.141,57.389,-30.648
C05220=1012.915,255.412,-142.663,-29.142,57.400,-30.649
C05221=1012.919,255.657,-142.692,-29.143,57.411,-30.648
C05222=1012.922,255.903,-142.721,-29.144,57.421,-30.647
C05223=1012.925,256.148,-142.750,-29.145,57.429,-30.646
C05224=1012.928,256.393,-142.779,-29.146,57.439,-30.646
C05225=1012.932,256.638,-142.808,-29.147,57.448,-30.647
C05226=1012.935,256.883,-142.837,-29.148,57.458,-30.645
C05227=1012.938,257.128,-142.866,-29.149,57.467,-30.645
C05228=1012.941,257.373,-142.895,-29.150,57.478,-30.645
C05229=1012.944,257.618,-142.923,-29.151,57.488,-30.644
C05230=1012.948,257.863,-142.952,-29.152,57.498,-30.643
C05231=1012.951,258.108,-142.981,-29.153,57.510,-30.644
C05232=1012.954,258.354,-143.011,-29.155,57.521,-30.643
C05233=1012.967,259.583,-143.163,-28.902,57.750,-29.618
C05234=1012.970,259.988,-143.217,-28.814,57.810,-29.274
C05235=1012.970,260.395,-143.270,-28.728,57.908,-28.927
C05236=1012.971,260.801,-143.327,-28.639,57.985,-28.579
C05237=1012.971,261.207,-143.384,-28.549,58.058,-28.230
C05238=1012.969,261.613,-143.442,-28.459,58.171,-27.876
C05239=1012.967,262.019,-143.502,-28.366,58.245,-27.523
C05240=1012.964,262.425,-143.563,-28.273,58.338,-27.168
C05241=1012.960,262.830,-143.627,-28.177,58.403,-26.812
C05242=1012.954,263.236,-143.691,-28.081,58.505,-26.452
C05243=1012.948,263.641,-143.757,-27.983,58.574,-26.094
C05244=1012.941,264.046,-143.824,-27.884,58.657,-25.732
C05245=1012.932,264.452,-143.892,-27.783,58.772,-25.366
C05246=1012.923,264.856,-143.962,-27.681,58.831,-25.004
C05247=1012.913,265.262,-144.034,-27.577,58.929,-24.635
C05248=1012.901,265.667,-144.105,-27.472,59.032,-24.266
C05249=1012.890,266.072,-144.180,-27.366,59.121,-23.896
C05250=1012.877,266.477,-144.256,-27.258,59.201,-23.524
C05251=1012.863,266.880,-144.332,-27.148,59.289,-23.149
C05252=1012.848,267.285,-144.411,-27.036,59.393,-22.771
C05253=1012.833,267.689,-144.491,-26.923,59.463,-22.392
C05254=1012.815,268.093,-144.572,-26.807,59.571,-22.010
C05255=1012.798,268.497,-144.655,-26.690,59.660,-21.626
C05256=1012.779,268.901,-144.740,-26.572,59.744,-21.241
C05257=1012.759,269.304,-144.824,-26.449,59.868,-20.848
C05258=1012.738,269.707,-144.911,-26.327,59.954,-20.459
C05259=1012.716,270.110,-144.999,-26.201,60.061,-20.064
C05260=1012.693,270.514,-145.090,-26.077,60.136,-19.670
C05261=1012.669,270.916,-145.181,-25.946,60.250,-19.269
C05262=1012.645,271.318,-145.273,-25.816,60.338,-18.869
C05263=1012.619,271.721,-145.368,-25.682,60.439,-18.465
C05264=1012.591,272.123,-145.464,-25.547,60.545,-18.058
C05265=1012.564,272.525,-145.561,-25.410,60.636,-17.649
C05266=1012.534,272.927,-145.658,-25.266,60.764,-17.233
C05267=1012.505,273.329,-145.759,-25.124,60.857,-16.818
C05268=1012.474,273.730,-145.862,-24.979,60.956,-16.398
C05269=1012.442,274.131,-145.964,-24.831,61.059,-15.975
C05270=1012.409,274.532,-146.068,-24.677,61.177,-15.545
C05271=1012.387,274.781,-146.134,-24.581,61.247,-15.277
C05272=1012.366,275.030,-146.201,-24.485,61.305,-15.008
C05273=1012.342,275.306,-146.275,-24.376,61.378,-14.706
C05274=1012.317,275.582,-146.350,-24.264,61.464,-14.403
C05275=1012.291,275.858,-146.425,-24.154,61.528,-14.099
C05276=1012.265,276.134,-146.502,-24.039,61.610,-13.791
C05277=1012.227,276.533,-146.614,-23.871,61.724,-13.342
C05278=1012.188,276.933,-146.728,-23.700,61.834,-12.889
C05279=1012.147,277.332,-146.842,-23.523,61.958,-12.428
C05280=1012.106,277.731,-146.961,-23.349,62.052,-11.970
C05281=1012.063,278.130,-147.078,-23.163,62.185,-11.500
C05282=1012.019,278.528,-147.198,-22.977,62.303,-11.028
C05283=1011.974,278.925,-147.320,-22.790,62.409,-10.552
C05284=1011.928,279.323,-147.443,-22.594,62.535,-10.070
C05285=1011.881,279.721,-147.567,-22.397,62.652,-9.582
C05286=1011.833,280.118,-147.693,-22.191,62.781,-9.085
C05287=1011.783,280.514,-147.821,-21.979,62.911,-8.580
C05288=1011.732,280.910,-147.951,-21.763,63.040,-8.068
C05289=1011.681,281.306,-148.082,-21.543,63.163,-7.549
C05290=1011.628,281.701,-148.214,-21.313,63.304,-7.021
C05291=1011.573,282.096,-148.348,-21.079,63.436,-6.486
C05292=1011.519,282.491,-148.484,-20.838,63.573,-5.940
C05293=1011.462,282.885,-148.622,-20.593,63.706,-5.389
C05294=1011.405,283.279,-148.761,-20.340,63.841,-4.828
C05295=1011.345,283.672,-148.902,-20.075,63.993,-4.255
C05296=1011.285,284.065,-149.044,-19.806,64.134,-3.676
C05297=1011.225,284.458,-149.189,-19.532,64.274,-3.087
C05298=1011.162,284.849,-149.336,-19.254,64.408,-2.492
C05299=1011.131,285.045,-149.410,-19.108,64.484,-2.188
C05300=1011.067,285.436,-149.558,-18.806,64.644,-1.571
C05301=1011.033,285.632,-149.632,-18.653,64.722,-1.259
C05302=1011.001,285.826,-149.708,-18.499,64.795,-0.944
C05303=1010.967,286.021,-149.784,-18.342,64.872,-0.625
C05304=1010.934,286.217,-149.861,-18.182,64.950,-0.303
C05305=1010.899,286.411,-149.937,-18.026,65.016,0.018
C05306=1010.866,286.606,-150.015,-17.861,65.094,0.347
C05307=1010.831,286.801,-150.092,-17.685,65.186,0.685
C05308=1010.796,286.995,-150.170,-17.518,65.259,1.020
C05309=1010.761,287.189,-150.249,-17.348,65.332,1.356
C05310=1010.725,287.383,-150.328,-17.169,65.418,1.700
C05311=1010.689,287.577,-150.407,-16.981,65.512,2.052
C05312=1010.653,287.771,-150.488,-16.802,65.588,2.401
C05313=1010.616,287.965,-150.568,-16.613,65.676,2.758
C05314=1010.580,288.157,-150.649,-16.428,65.751,3.114
C05315=1010.542,288.350,-150.730,-16.239,65.830,3.474
C05316=1010.505,288.544,-150.811,-16.038,65.922,3.843
C05317=1010.467,288.737,-150.894,-15.835,66.011,4.217
///RCONF 0,0,0,0,0,0,0,0,0,0,0,0,0,0,0,0,0,0,0,0,0,0,0,0
C05318=1010.428,288.929,-150.977,-15.632,66.098,4.590
C05319=1010.390,289.122,-151.061,-15.428,66.180,4.969
C05320=1010.351,289.314,-151.144,-15.217,66.268,5.352
C05321=1010.311,289.507,-151.228,-15.005,66.352,5.740
C05322=1010.272,289.698,-151.312,-14.786,66.440,6.133
C05323=1010.232,289.890,-151.398,-14.561,66.532,6.533
C05324=1010.192,290.082,-151.484,-14.341,66.613,6.932
C05325=1010.151,290.273,-151.570,-14.105,66.707,7.345
C05326=1010.110,290.464,-151.656,-13.872,66.795,7.757
C05327=1010.069,290.656,-151.744,-13.634,66.882,8.175
C05328=1010.026,290.846,-151.832,-13.382,66.982,8.604
C05329=1009.985,291.037,-151.919,-13.135,67.071,9.033
C05330=1009.942,291.228,-152.009,-12.878,67.167,9.470
C05331=1009.899,291.417,-152.098,-12.627,67.252,9.907
C05332=1009.855,291.607,-152.187,-12.358,67.349,10.358
C05333=1009.812,291.797,-152.278,-12.096,67.435,10.806
C05334=1009.768,291.986,-152.369,-11.827,67.523,11.262
C05335=1009.724,292.176,-152.460,-11.540,67.626,11.732
C05336=1009.678,292.365,-152.552,-11.252,67.724,12.205
C05337=1009.633,292.554,-152.644,-10.959,67.821,12.686
C05338=1009.588,292.742,-152.737,-10.665,67.913,13.168
C05339=1009.542,292.931,-152.830,-10.361,68.011,13.661
C05340=1009.496,293.119,-152.925,-10.054,68.105,14.159
C05341=1009.449,293.307,-153.019,-9.740,68.200,14.664
C05342=1009.401,293.495,-153.114,-9.412,68.302,15.182
C05343=1009.354,293.683,-153.210,-9.090,68.394,15.699
C05344=1009.306,293.869,-153.306,-8.746,68.498,16.234
C05345=1009.258,294.056,-153.403,-8.411,68.590,16.765
C05346=1009.209,294.243,-153.500,-8.060,68.690,17.310
C05347=1009.160,294.429,-153.598,-7.699,68.791,17.866
C05348=1009.110,294.616,-153.696,-7.331,68.893,18.429
C05349=1009.061,294.801,-153.796,-6.967,68.985,18.994
C05350=1009.010,294.987,-153.895,-6.581,69.089,19.576
C05351=1008.960,295.172,-153.996,-6.206,69.178,20.152
C05352=1008.908,295.358,-154.097,-5.813,69.276,20.745
C05353=1008.857,295.542,-154.197,-5.392,69.387,21.361
C05354=1008.804,295.727,-154.299,-4.984,69.483,21.972
C05355=1008.752,295.911,-154.402,-4.564,69.581,22.594
C05356=1008.699,296.095,-154.505,-4.135,69.679,23.224
C05357=1008.646,296.278,-154.609,-3.699,69.776,23.864
C05358=1008.592,296.462,-154.712,-3.250,69.875,24.517
C05359=1008.538,296.644,-154.817,-2.794,69.971,25.178
C05360=1008.483,296.827,-154.923,-2.331,70.067,25.846
C05361=1008.428,297.010,-155.028,-1.847,70.169,26.533
C05362=1008.373,297.191,-155.136,-1.374,70.257,27.217
C05363=1008.317,297.374,-155.243,-0.872,70.357,27.924
C05364=1008.260,297.555,-155.351,-0.360,70.455,28.642
C05365=1008.203,297.736,-155.460,0.146,70.544,29.358
C05366=1008.146,297.917,-155.568,0.687,70.646,30.105
C05367=1008.088,298.097,-155.678,1.228,70.740,30.854
C05368=1008.029,298.278,-155.788,1.785,70.836,31.618
C05369=1007.971,298.458,-155.899,2.330,70.920,32.376
